DATA_BLOCK DB 5
AUTHOR : NUMERIK
FAMILY : _800D
NAME : Basics
VERSION : 1.5
  STRUCT
   Ch1_DB2_310 : BOOL  := TRUE;	// (Channel 1-10 ever 18 Bits):  error message
   Ch1_DB2_311 : BOOL ;	// Channel 1, DB2.DBB311; operational message
   Ch1_DB2_312 : BOOL  := TRUE;	// Channel 1, DB2.DBB312; error message
   Ch1_DB2_313 : BOOL  := TRUE;	// error message
   Ch1_DB2_314 : BOOL ;	// operational message
   Ch1_DB2_315 : BOOL ;	// operational message
   Ch1_DB2_316 : BOOL  := TRUE;	// error message
   Ch1_DB2_317 : BOOL  := TRUE;	// error message
   Ch1_DB2_318 : BOOL ;	// operational message
   Ch1_DB2_319 : BOOL ;	// operational message
   Ch1_DB2_320 : BOOL  := TRUE;	// error message
   Ch1_DB2_321 : BOOL ;	// operational message
   Ch1_DB2_322 : BOOL  := TRUE;	// error message
   Ch1_DB2_323 : BOOL ;	// operational message
   Ch1_DB2_324 : BOOL  := TRUE;	// error message
   Ch1_DB2_325 : BOOL ;	// operational message
   Ch1_DB2_326 : BOOL  := TRUE;	// error message
   Ch1_DB2_327 : BOOL ;	// operational message
   Ch2_DB2_328 : BOOL  := TRUE;	// Channel 2, DB2.DBB328; error message
   Ch2_DB2_329 : BOOL ;	// Channel 2, DB2.DBB329; operational message
   Ch2_DB2_330 : BOOL  := TRUE;	// error message
   Ch2_DB2_331 : BOOL  := TRUE;	// error message
   Ch2_DB2_332 : BOOL ;	// operational message
   Ch2_DB2_333 : BOOL ;	// operational message
   Ch2_DB2_334 : BOOL  := TRUE;	// error message
   Ch2_DB2_335 : BOOL  := TRUE;	// error message
   Ch2_DB2_336 : BOOL ;	// operational message
   Ch2_DB2_337 : BOOL ;	// operational message
   Ch2_DB2_338 : BOOL  := TRUE;	// error message
   Ch2_DB2_339 : BOOL ;	// operational message
   Ch2_DB2_340 : BOOL  := TRUE;	// error message
   Ch2_DB2_341 : BOOL ;	// operational message
   Ch2_DB2_342 : BOOL  := TRUE;	// error message
   Ch2_DB2_343 : BOOL ;	// operational message
   Ch2_DB2_344 : BOOL  := TRUE;	// error message
   Ch2_DB2_345 : BOOL ;	// operational message
   Ch3_DB2_346 : BOOL  := TRUE;	// Channel 3, DB2.DBB346; error message
   Ch3_DB2_347 : BOOL ;	// Channel 3, DB2.DBB347; operational message
   Ch3_DB2_348 : BOOL  := TRUE;	// error message
   Ch3_DB2_349 : BOOL  := TRUE;	// error message
   Ch3_DB2_350 : BOOL ;	// operational message
   Ch3_DB2_351 : BOOL ;	// operational message
   Ch3_DB2_352 : BOOL  := TRUE;	// error message
   Ch3_DB2_353 : BOOL  := TRUE;	// error message
   Ch3_DB2_354 : BOOL ;	// operational message
   Ch3_DB2_355 : BOOL ;	// operational message
   Ch3_DB2_356 : BOOL  := TRUE;	// error message
   Ch3_DB2_357 : BOOL ;	// operational message
   Ch3_DB2_358 : BOOL  := TRUE;	// error message
   Ch3_DB2_359 : BOOL ;	// operational message
   Ch3_DB2_360 : BOOL  := TRUE;	// error message
   Ch3_DB2_361 : BOOL ;	// operational message
   Ch3_DB2_362 : BOOL  := TRUE;	// error message
   Ch3_DB2_363 : BOOL ;	// operational message
   Ch4_DB2_364 : BOOL  := TRUE;	// Channel 4, DB2.DBB364; error message
   Ch4_DB2_365 : BOOL ;	// Channel 4, DB2.DBB365; operational message
   Ch4_DB2_366 : BOOL  := TRUE;	// error message
   Ch4_DB2_367 : BOOL  := TRUE;	// error message
   Ch4_DB2_368 : BOOL ;	// operational message
   Ch4_DB2_369 : BOOL ;	// operational message
   Ch4_DB2_370 : BOOL  := TRUE;	// error message
   Ch4_DB2_371 : BOOL  := TRUE;	// error message
   Ch4_DB2_372 : BOOL ;	// operational message
   Ch4_DB2_373 : BOOL ;	// operational message
   Ch4_DB2_374 : BOOL  := TRUE;	// error message
   Ch4_DB2_375 : BOOL ;	// operational message
   Ch4_DB2_376 : BOOL  := TRUE;	// error message
   Ch4_DB2_377 : BOOL ;	// operational message
   Ch4_DB2_378 : BOOL  := TRUE;	// error message
   Ch4_DB2_379 : BOOL ;	// operational message
   Ch4_DB2_380 : BOOL  := TRUE;	// error message
   Ch4_DB2_381 : BOOL ;	// operational message
   Ch5_DB2_382 : BOOL  := TRUE;	// Channel 5, DB2.DBB382; error message
   Ch5_DB2_383 : BOOL ;	// Channel 5, DB2.DBB383; operational message
   Ch5_DB2_384 : BOOL  := TRUE;	// error message
   Ch5_DB2_385 : BOOL  := TRUE;	// error message
   Ch5_DB2_386 : BOOL ;	// operational message
   Ch5_DB2_387 : BOOL ;	// operational message
   Ch5_DB2_388 : BOOL  := TRUE;	// error message
   Ch5_DB2_389 : BOOL  := TRUE;	// error message
   Ch5_DB2_390 : BOOL ;	// operational message
   Ch5_DB2_391 : BOOL ;	// operational message
   Ch5_DB2_392 : BOOL  := TRUE;	// error message
   Ch5_DB2_393 : BOOL ;	// operational message
   Ch5_DB2_394 : BOOL  := TRUE;	// error message
   Ch5_DB2_395 : BOOL ;	// operational message
   Ch5_DB2_396 : BOOL  := TRUE;	// error message
   Ch5_DB2_397 : BOOL ;	// operational message
   Ch5_DB2_398 : BOOL  := TRUE;	// error message
   Ch5_DB2_399 : BOOL ;	// operational message
   Ch6_DB2_400 : BOOL  := TRUE;	// Channel 6, DB2.DBB400; error message
   Ch6_DB2_401 : BOOL ;	// Channel 6, DB2.DBB401; operational message
   Ch6_DB2_402 : BOOL  := TRUE;	// error message
   Ch6_DB2_403 : BOOL  := TRUE;	// error message
   Ch6_DB2_404 : BOOL ;	// operational message
   Ch6_DB2_405 : BOOL ;	// operational message
   Ch6_DB2_406 : BOOL  := TRUE;	// error message
   Ch6_DB2_407 : BOOL  := TRUE;	// error message
   Ch6_DB2_408 : BOOL ;	// operational message
   Ch6_DB2_409 : BOOL ;	// operational message
   Ch6_DB2_410 : BOOL  := TRUE;	// error message
   Ch6_DB2_411 : BOOL ;	// operational message
   Ch6_DB2_412 : BOOL  := TRUE;	// error message
   Ch6_DB2_413 : BOOL ;	// operational message
   Ch6_DB2_414 : BOOL  := TRUE;	// error message
   Ch6_DB2_415 : BOOL ;	// operational message
   Ch6_DB2_416 : BOOL  := TRUE;	// error message
   Ch6_DB2_417 : BOOL ;	// operational message
   Ch7_DB2_418 : BOOL  := TRUE;	// Channel 7, DB2.DBB418; error message
   Ch7_DB2_419 : BOOL ;	// Channel 7, DB2.DBB419; operational message
   Ch7_DB2_420 : BOOL  := TRUE;	// error message
   Ch7_DB2_421 : BOOL  := TRUE;	// error message
   Ch7_DB2_422 : BOOL ;	// operational message
   Ch7_DB2_423 : BOOL ;	// operational message
   Ch7_DB2_424 : BOOL  := TRUE;	// error message
   Ch7_DB2_425 : BOOL  := TRUE;	// error message
   Ch7_DB2_426 : BOOL ;	// operational message
   Ch7_DB2_427 : BOOL ;	// operational message
   Ch7_DB2_428 : BOOL  := TRUE;	// error message
   Ch7_DB2_429 : BOOL ;	// operational message
   Ch7_DB2_430 : BOOL  := TRUE;	// error message
   Ch7_DB2_431 : BOOL ;	// operational message
   Ch7_DB2_432 : BOOL  := TRUE;	// error message
   Ch7_DB2_433 : BOOL ;	// operational message
   Ch7_DB2_434 : BOOL  := TRUE;	// error message
   Ch7_DB2_435 : BOOL ;	// operational message
   Ch8_DB2_436 : BOOL  := TRUE;	// Channel 8, DB2.DBB436; error message
   Ch8_DB2_437 : BOOL ;	// Channel 8, DB2.DBB437; operational message
   Ch8_DB2_438 : BOOL  := TRUE;	// error message
   Ch8_DB2_439 : BOOL  := TRUE;	// error message
   Ch8_DB2_440 : BOOL ;	// operational message
   Ch8_DB2_441 : BOOL ;	// operational message
   Ch8_DB2_442 : BOOL  := TRUE;	// error message
   Ch8_DB2_443 : BOOL  := TRUE;	// error message
   Ch8_DB2_444 : BOOL ;	// operational message
   Ch8_DB2_445 : BOOL ;	// operational message
   Ch8_DB2_446 : BOOL  := TRUE;	// error message
   Ch8_DB2_447 : BOOL ;	// operational message
   Ch8_DB2_448 : BOOL  := TRUE;	// error message
   Ch8_DB2_449 : BOOL ;	// operational message
   Ch8_DB2_450 : BOOL  := TRUE;	// error message
   Ch8_DB2_451 : BOOL ;	// operational message
   Ch8_DB2_452 : BOOL  := TRUE;	// error message
   Ch8_DB2_453 : BOOL ;	// operational message
   Ch9_DB2_454 : BOOL  := TRUE;	// Channel 9, DB2.DBB454; error message
   Ch9_DB2_455 : BOOL ;	// Channel 9, DB2.DBB455; operational message
   Ch9_DB2_456 : BOOL  := TRUE;	// error message
   Ch9_DB2_457 : BOOL  := TRUE;	// error message
   Ch9_DB2_458 : BOOL ;	// operational message
   Ch9_DB2_459 : BOOL ;	// operational message
   Ch9_DB2_460 : BOOL  := TRUE;	// error message
   Ch9_DB2_461 : BOOL  := TRUE;	// error message
   Ch9_DB2_462 : BOOL ;	// operational message
   Ch9_DB2_463 : BOOL ;	// operational message
   Ch9_DB2_464 : BOOL  := TRUE;	// error message
   Ch9_DB2_465 : BOOL ;	// operational message
   Ch9_DB2_466 : BOOL  := TRUE;	// error message
   Ch9_DB2_467 : BOOL ;	// operational message
   Ch9_DB2_468 : BOOL  := TRUE;	// error message
   Ch9_DB2_469 : BOOL ;	// operational message
   Ch9_DB2_470 : BOOL  := TRUE;	// error message
   Ch9_DB2_471 : BOOL ;	// operational message
   Ch10_DB2_472 : BOOL  := TRUE;	// Channel 10, DB2.DBB472; error message
   Ch10_DB2_473 : BOOL ;	// Channel 10, DB2.DBB473; operational message
   Ch10_DB2_474 : BOOL  := TRUE;	// error message
   Ch10_DB2_475 : BOOL  := TRUE;	// error message
   Ch10_DB2_476 : BOOL ;	// operational message
   Ch10_DB2_477 : BOOL ;	// operational message
   Ch10_DB2_478 : BOOL  := TRUE;	// error message
   Ch10_DB2_479 : BOOL  := TRUE;	// error message
   Ch10_DB2_480 : BOOL ;	// operational message
   Ch10_DB2_481 : BOOL ;	// operational message
   Ch10_DB2_482 : BOOL  := TRUE;	// error message
   Ch10_DB2_483 : BOOL ;	// operational message
   Ch10_DB2_484 : BOOL  := TRUE;	// error message
   Ch10_DB2_485 : BOOL ;	// operational message
   Ch10_DB2_486 : BOOL  := TRUE;	// error message
   Ch10_DB2_487 : BOOL ;	// operational message
   Ch10_DB2_488 : BOOL  := TRUE;	// error message
   Ch10_DB2_489 : BOOL ;	// operational message
   Ax1_DB2_490 : BOOL  := TRUE;	// (32 Axes/Spindles ever 2 Bit):  error message
   Ax1_DB2_491 : BOOL ;	// Axis 1, DB2.DBB491; operational message
   Ax2_DB2_492 : BOOL  := TRUE;	// Axis 2, DB2.DBB492; error message
   Ax2_DB2_493 : BOOL ;	// Axis 2, DB2.DBB493; operational message
   Ax3_DB2_494 : BOOL  := TRUE;	// error message
   Ax3_DB2_495 : BOOL ;	// operational message
   Ax4_DB2_496 : BOOL  := TRUE;	// error message
   Ax4_DB2_497 : BOOL ;	// operational message
   Ax5_DB2_498 : BOOL  := TRUE;	// error message
   Ax5_DB2_499 : BOOL ;	// operational message
   Ax6_DB2_500 : BOOL  := TRUE;	// error message
   Ax6_DB2_501 : BOOL ;	// operational message
   Ax7_DB2_502 : BOOL  := TRUE;	// error message
   Ax7_DB2_503 : BOOL ;	// operational message
   Ax8_DB2_504 : BOOL  := TRUE;	// error message
   Ax8_DB2_505 : BOOL ;	// operational message
   Ax9_DB2_506 : BOOL  := TRUE;	// error message
   Ax9_DB2_507 : BOOL ;	// operational message
   Ax10_DB2_508 : BOOL  := TRUE;	// error message
   Ax10_DB2_509 : BOOL ;	// operational message
   Ax11_DB2_510 : BOOL  := TRUE;	// error message
   Ax11_DB2_511 : BOOL ;	// operational message
   Ax12_DB2_512 : BOOL  := TRUE;	// error message
   Ax12_DB2_513 : BOOL ;	// operational message
   Ax13_DB2_514 : BOOL  := TRUE;	// error message
   Ax13_DB2_515 : BOOL ;	// operational message
   Ax14_DB2_516 : BOOL  := TRUE;	// error message
   Ax14_DB2_517 : BOOL ;	// operational message
   Ax15_DB2_518 : BOOL  := TRUE;	// error message
   Ax15_DB2_519 : BOOL ;	// operational message
   Ax16_DB2_520 : BOOL  := TRUE;	// error message
   Ax16_DB2_521 : BOOL ;	// operational message
   Ax17_DB2_522 : BOOL  := TRUE;	// error message
   Ax17_DB2_523 : BOOL ;	// operational message
   Ax18_DB2_524 : BOOL  := TRUE;	// error message
   Ax18_DB2_525 : BOOL ;	// operational message
   Ax19_DB2_526 : BOOL  := TRUE;	// error message
   Ax19_DB2_527 : BOOL ;	// operational message
   Ax20_DB2_528 : BOOL  := TRUE;	// error message
   Ax20_DB2_529 : BOOL ;	// operational message
   Ax21_DB2_530 : BOOL  := TRUE;	// error message
   Ax21_DB2_531 : BOOL ;	// operational message
   Ax22_DB2_532 : BOOL  := TRUE;	// error message
   Ax22_DB2_533 : BOOL ;	// operational message
   Ax23_DB2_534 : BOOL  := TRUE;	// error message
   Ax23_DB2_535 : BOOL ;	// operational message
   Ax24_DB2_536 : BOOL  := TRUE;	// error message
   Ax24_DB2_537 : BOOL ;	// operational message
   Ax25_DB2_538 : BOOL  := TRUE;	// error message
   Ax25_DB2_539 : BOOL ;	// operational message
   Ax26_DB2_540 : BOOL  := TRUE;	// error message
   Ax26_DB2_541 : BOOL ;	// operational message
   Ax27_DB2_542 : BOOL  := TRUE;	// error message
   Ax27_DB2_543 : BOOL ;	// operational message
   Ax28_DB2_544 : BOOL  := TRUE;	// error message
   Ax28_DB2_545 : BOOL ;	// operational message
   Ax29_DB2_546 : BOOL  := TRUE;	// error message
   Ax29_DB2_547 : BOOL ;	// operational message
   Ax30_DB2_548 : BOOL  := TRUE;	// error message
   Ax30_DB2_549 : BOOL ;	// operational message
   Ax31_DB2_550 : BOOL  := TRUE;	// error message
   Ax31_DB2_551 : BOOL ;	// operational message
   Ax32_DB2_552 : BOOL  := TRUE;	// error message
   Ax32_DB2_553 : BOOL ;	// operational message
   User0_DB2_554 : BOOL  := TRUE;	// (32 User data area ever 8 Bit):  error message
   User0_DB2_555 : BOOL  := TRUE;	// UserDataArea 0, DB2.DBB555; error message
   User0_DB2_556 : BOOL  := TRUE;	// error message
   User0_DB2_557 : BOOL  := TRUE;	// error message
   User0_DB2_558 : BOOL ;	// operational message
   User0_DB2_559 : BOOL ;	// operational message
   User0_DB2_560 : BOOL ;	// operational message
   User0_DB2_561 : BOOL ;	// operational message
   User1_DB2_562 : BOOL  := TRUE;	// UserDataArea 1, DB2.DBB562; error message
   User1_DB2_563 : BOOL  := TRUE;	// error message
   User1_DB2_564 : BOOL  := TRUE;	// error message
   User1_DB2_565 : BOOL  := TRUE;	// error message
   User1_DB2_566 : BOOL ;	// operational message
   User1_DB2_567 : BOOL ;	// operational message
   User1_DB2_568 : BOOL ;	// operational message
   User1_DB2_569 : BOOL ;	// operational message
   User2_DB2_570 : BOOL  := TRUE;	// UserDataArea 2, DB2.DBB570; error message
   User2_DB2_571 : BOOL  := TRUE;	// error message
   User2_DB2_572 : BOOL  := TRUE;	// error message
   User2_DB2_573 : BOOL  := TRUE;	// error message
   User2_DB2_574 : BOOL ;	// operational message
   User2_DB2_575 : BOOL ;	// operational message
   User2_DB2_576 : BOOL ;	// operational message
   User2_DB2_577 : BOOL ;	// operational message
   User3_DB2_578 : BOOL  := TRUE;	// UserDataArea 3, DB2.DBB578; error message
   User3_DB2_579 : BOOL  := TRUE;	// error message
   User3_DB2_580 : BOOL  := TRUE;	// error message
   User3_DB2_581 : BOOL  := TRUE;	// error message
   User3_DB2_582 : BOOL ;	// operational message
   User3_DB2_583 : BOOL ;	// operational message
   User3_DB2_584 : BOOL ;	// operational message
   User3_DB2_585 : BOOL ;	// operational message
   User4_DB2_586 : BOOL  := TRUE;	// UserDataArea 4, DB2.DBB586; error message
   User4_DB2_587 : BOOL  := TRUE;	// error message
   User4_DB2_588 : BOOL  := TRUE;	// error message
   User4_DB2_589 : BOOL  := TRUE;	// error message
   User4_DB2_590 : BOOL ;	// operational message
   User4_DB2_591 : BOOL ;	// operational message
   User4_DB2_592 : BOOL ;	// operational message
   User4_DB2_593 : BOOL ;	// operational message
   User5_DB2_594 : BOOL  := TRUE;	// UserDataArea 5, DB2.DBB594; error message
   User5_DB2_595 : BOOL  := TRUE;	// error message
   User5_DB2_596 : BOOL  := TRUE;	// error message
   User5_DB2_597 : BOOL  := TRUE;	// error message
   User5_DB2_598 : BOOL ;	// operational message
   User5_DB2_599 : BOOL ;	// operational message
   User5_DB2_600 : BOOL ;	// operational message
   User5_DB2_601 : BOOL ;	// operational message
   User6_DB2_602 : BOOL  := TRUE;	// UserDataArea 6, DB2.DBB602; error message
   User6_DB2_603 : BOOL  := TRUE;	// error message
   User6_DB2_604 : BOOL  := TRUE;	// error message
   User6_DB2_605 : BOOL  := TRUE;	// error message
   User6_DB2_606 : BOOL ;	// operational message
   User6_DB2_607 : BOOL ;	// operational message
   User6_DB2_608 : BOOL ;	// operational message
   User6_DB2_609 : BOOL ;	// operational message
   User7_DB2_610 : BOOL  := TRUE;	// UserDataArea 7, DB2.DBB610; error message
   User7_DB2_611 : BOOL  := TRUE;	// error message
   User7_DB2_612 : BOOL  := TRUE;	// error message
   User7_DB2_613 : BOOL  := TRUE;	// error message
   User7_DB2_614 : BOOL ;	// operational message
   User7_DB2_615 : BOOL ;	// operational message
   User7_DB2_616 : BOOL ;	// operational message
   User7_DB2_617 : BOOL ;	// operational message
   User8_DB2_618 : BOOL  := TRUE;	// UserDataArea 8, DB2.DBB618; error message
   User8_DB2_619 : BOOL  := TRUE;	// error message
   User8_DB2_620 : BOOL  := TRUE;	// error message
   User8_DB2_621 : BOOL  := TRUE;	// error message
   User8_DB2_622 : BOOL ;	// operational message
   User8_DB2_623 : BOOL ;	// operational message
   User8_DB2_624 : BOOL ;	// operational message
   User8_DB2_625 : BOOL ;	// operational message
   User9_DB2_626 : BOOL  := TRUE;	// UserDataArea 9, DB2.DBB626; error message
   User9_DB2_627 : BOOL  := TRUE;	// error message
   User9_DB2_628 : BOOL  := TRUE;	// error message
   User9_DB2_629 : BOOL  := TRUE;	// error message
   User9_DB2_630 : BOOL ;	// operational message
   User9_DB2_631 : BOOL ;	// operational message
   User9_DB2_632 : BOOL ;	// operational message
   User9_DB2_633 : BOOL ;	// operational message
   User10_DB2_634 : BOOL  := TRUE;	// UserDataArea 10, DB2.DBB634; error message
   User10_DB2_635 : BOOL  := TRUE;	// error message
   User10_DB2_636 : BOOL  := TRUE;	// error message
   User10_DB2_637 : BOOL  := TRUE;	// error message
   User10_DB2_638 : BOOL ;	// operational message
   User10_DB2_639 : BOOL ;	// operational message
   User10_DB2_640 : BOOL ;	// operational message
   User10_DB2_641 : BOOL ;	// operational message
   User11_DB2_642 : BOOL  := TRUE;	// UserDataArea 11, DB2.DBB642; error message
   User11_DB2_643 : BOOL  := TRUE;	// error message
   User11_DB2_644 : BOOL  := TRUE;	// error message
   User11_DB2_645 : BOOL  := TRUE;	// error message
   User11_DB2_646 : BOOL ;	// operational message
   User11_DB2_647 : BOOL ;	// operational message
   User11_DB2_648 : BOOL ;	// operational message
   User11_DB2_649 : BOOL ;	// operational message
   User12_DB2_650 : BOOL  := TRUE;	// UserDataArea 12, DB2.DBB650; error message
   User12_DB2_651 : BOOL  := TRUE;	// error message
   User12_DB2_652 : BOOL  := TRUE;	// error message
   User12_DB2_653 : BOOL  := TRUE;	// error message
   User12_DB2_654 : BOOL ;	// operational message
   User12_DB2_655 : BOOL ;	// operational message
   User12_DB2_656 : BOOL ;	// operational message
   User12_DB2_657 : BOOL ;	// operational message
   User13_DB2_658 : BOOL  := TRUE;	// UserDataArea 13, DB2.DBB658; error message
   User13_DB2_659 : BOOL  := TRUE;	// error message
   User13_DB2_660 : BOOL  := TRUE;	// error message
   User13_DB2_661 : BOOL  := TRUE;	// error message
   User13_DB2_662 : BOOL ;	// operational message
   User13_DB2_663 : BOOL ;	// operational message
   User13_DB2_664 : BOOL ;	// operational message
   User13_DB2_665 : BOOL ;	// operational message
   User14_DB2_666 : BOOL  := TRUE;	// UserDataArea 14, DB2.DBB666; error message
   User14_DB2_667 : BOOL  := TRUE;	// error message
   User14_DB2_668 : BOOL  := TRUE;	// error message
   User14_DB2_669 : BOOL  := TRUE;	// error message
   User14_DB2_670 : BOOL ;	// operational message
   User14_DB2_671 : BOOL ;	// operational message
   User14_DB2_672 : BOOL ;	// operational message
   User14_DB2_673 : BOOL ;	// operational message
   User15_DB2_674 : BOOL  := TRUE;	// UserDataArea 15, DB2.DBB674; error message
   User15_DB2_675 : BOOL  := TRUE;	// error message
   User15_DB2_676 : BOOL  := TRUE;	// error message
   User15_DB2_677 : BOOL  := TRUE;	// error message
   User15_DB2_678 : BOOL ;	// operational message
   User15_DB2_679 : BOOL ;	// operational message
   User15_DB2_680 : BOOL ;	// operational message
   User15_DB2_681 : BOOL ;	// operational message
   User16_DB2_682 : BOOL  := TRUE;	// UserDataArea 16, DB2.DBB682; error message
   User16_DB2_683 : BOOL  := TRUE;	// error message
   User16_DB2_684 : BOOL  := TRUE;	// error message
   User16_DB2_685 : BOOL  := TRUE;	// error message
   User16_DB2_686 : BOOL ;	// operational message
   User16_DB2_687 : BOOL ;	// operational message
   User16_DB2_688 : BOOL ;	// operational message
   User16_DB2_689 : BOOL ;	// operational message
   User17_DB2_690 : BOOL  := TRUE;	// UserDataArea 17, DB2.DBB690; error message
   User17_DB2_691 : BOOL  := TRUE;	// error message
   User17_DB2_692 : BOOL  := TRUE;	// error message
   User17_DB2_693 : BOOL  := TRUE;	// error message
   User17_DB2_694 : BOOL ;	// operational message
   User17_DB2_695 : BOOL ;	// operational message
   User17_DB2_696 : BOOL ;	// operational message
   User17_DB2_697 : BOOL ;	// operational message
   User18_DB2_698 : BOOL  := TRUE;	// UserDataArea 18, DB2.DBB698; error message
   User18_DB2_699 : BOOL  := TRUE;	// error message
   User18_DB2_700 : BOOL  := TRUE;	// error message
   User18_DB2_701 : BOOL  := TRUE;	// error message
   User18_DB2_702 : BOOL ;	// operational message
   User18_DB2_703 : BOOL ;	// operational message
   User18_DB2_704 : BOOL ;	// operational message
   User18_DB2_705 : BOOL ;	// operational message
   User19_DB2_706 : BOOL  := TRUE;	// UserDataArea 19, DB2.DBB706; error message
   User19_DB2_707 : BOOL  := TRUE;	// error message
   User19_DB2_708 : BOOL  := TRUE;	// error message
   User19_DB2_709 : BOOL  := TRUE;	// error message
   User19_DB2_710 : BOOL ;	// operational message
   User19_DB2_711 : BOOL ;	// operational message
   User19_DB2_712 : BOOL ;	// operational message
   User19_DB2_713 : BOOL ;	// operational message
   User20_DB2_714 : BOOL  := TRUE;	// UserDataArea 20, DB2.DBB714; error message
   User20_DB2_715 : BOOL  := TRUE;	// error message
   User20_DB2_716 : BOOL  := TRUE;	// error message
   User20_DB2_717 : BOOL  := TRUE;	// error message
   User20_DB2_718 : BOOL ;	// operational message
   User20_DB2_719 : BOOL ;	// operational message
   User20_DB2_720 : BOOL ;	// operational message
   User20_DB2_721 : BOOL ;	// operational message
   User21_DB2_722 : BOOL  := TRUE;	// UserDataArea 21, DB2.DBB722; error message
   User21_DB2_723 : BOOL  := TRUE;	// error message
   User21_DB2_724 : BOOL  := TRUE;	// error message
   User21_DB2_725 : BOOL  := TRUE;	// error message
   User21_DB2_726 : BOOL ;	// operational message
   User21_DB2_727 : BOOL ;	// operational message
   User21_DB2_728 : BOOL ;	// operational message
   User21_DB2_729 : BOOL ;	// operational message
   User22_DB2_730 : BOOL  := TRUE;	// UserDataArea 22, DB2.DBB730; error message
   User22_DB2_731 : BOOL  := TRUE;	// error message
   User22_DB2_732 : BOOL  := TRUE;	// error message
   User22_DB2_733 : BOOL  := TRUE;	// error message
   User22_DB2_734 : BOOL ;	// operational message
   User22_DB2_735 : BOOL ;	// operational message
   User22_DB2_736 : BOOL ;	// operational message
   User22_DB2_737 : BOOL ;	// operational message
   User23_DB2_738 : BOOL  := TRUE;	// UserDataArea 23, DB2.DBB738; error message
   User23_DB2_739 : BOOL  := TRUE;	// error message
   User23_DB2_740 : BOOL  := TRUE;	// error message
   User23_DB2_741 : BOOL  := TRUE;	// error message
   User23_DB2_742 : BOOL ;	// operational message
   User23_DB2_743 : BOOL ;	// operational message
   User23_DB2_744 : BOOL ;	// operational message
   User23_DB2_745 : BOOL ;	// operational message
   User24_DB2_746 : BOOL  := TRUE;	// UserDataArea 24, DB2.DBB746; error message
   User24_DB2_747 : BOOL  := TRUE;	// error message
   User24_DB2_748 : BOOL  := TRUE;	// error message
   User24_DB2_749 : BOOL  := TRUE;	// error message
   User24_DB2_750 : BOOL ;	// operational message
   User24_DB2_751 : BOOL ;	// operational message
   User24_DB2_752 : BOOL ;	// operational message
   User24_DB2_753 : BOOL ;	// operational message
   User25_DB2_754 : BOOL  := TRUE;	// UserDataArea 25, DB2.DBB754; error message
   User25_DB2_755 : BOOL  := TRUE;	// error message
   User25_DB2_756 : BOOL  := TRUE;	// error message
   User25_DB2_757 : BOOL  := TRUE;	// error message
   User25_DB2_758 : BOOL ;	// operational message
   User25_DB2_759 : BOOL ;	// operational message
   User25_DB2_760 : BOOL ;	// operational message
   User25_DB2_761 : BOOL ;	// operational message
   User26_DB2_762 : BOOL  := TRUE;	// UserDataArea 26, DB2.DBB762; error message
   User26_DB2_763 : BOOL  := TRUE;	// error message
   User26_DB2_764 : BOOL  := TRUE;	// error message
   User26_DB2_765 : BOOL  := TRUE;	// error message
   User26_DB2_766 : BOOL ;	// operational message
   User26_DB2_767 : BOOL ;	// operational message
   User26_DB2_768 : BOOL ;	// operational message
   User26_DB2_769 : BOOL ;	// operational message
   User27_DB2_770 : BOOL  := TRUE;	// UserDataArea 27, DB2.DBB770; error message
   User27_DB2_771 : BOOL  := TRUE;	// error message
   User27_DB2_772 : BOOL  := TRUE;	// error message
   User27_DB2_773 : BOOL  := TRUE;	// error message
   User27_DB2_774 : BOOL ;	// operational message
   User27_DB2_775 : BOOL ;	// operational message
   User27_DB2_776 : BOOL ;	// operational message
   User27_DB2_777 : BOOL ;	// operational message
   User28_DB2_778 : BOOL  := TRUE;	// UserDataArea 28, DB2.DBB778; error message
   User28_DB2_779 : BOOL  := TRUE;	// error message
   User28_DB2_780 : BOOL  := TRUE;	// error message
   User28_DB2_781 : BOOL  := TRUE;	// error message
   User28_DB2_782 : BOOL ;	// operational message
   User28_DB2_783 : BOOL ;	// operational message
   User28_DB2_784 : BOOL ;	// operational message
   User28_DB2_785 : BOOL ;	// operational message
   User29_DB2_786 : BOOL  := TRUE;	// UserDataArea 29, DB2.DBB786; error message
   User29_DB2_787 : BOOL  := TRUE;	// error message
   User29_DB2_788 : BOOL  := TRUE;	// error message
   User29_DB2_789 : BOOL  := TRUE;	// error message
   User29_DB2_790 : BOOL ;	// operational message
   User29_DB2_791 : BOOL ;	// operational message
   User29_DB2_792 : BOOL ;	// operational message
   User29_DB2_793 : BOOL ;	// operational message
   User30_DB2_794 : BOOL  := TRUE;	// UserDataArea 30, DB2.DBB794; error message
   User30_DB2_795 : BOOL  := TRUE;	// error message
   User30_DB2_796 : BOOL  := TRUE;	// error message
   User30_DB2_797 : BOOL  := TRUE;	// error message
   User30_DB2_798 : BOOL ;	// operational message
   User30_DB2_799 : BOOL ;	// operational message
   User30_DB2_800 : BOOL ;	// operational message
   User30_DB2_801 : BOOL ;	// operational message
   User31_DB2_802 : BOOL  := TRUE;	// UserDataArea 31, DB2.DBB802; error message
   User31_DB2_803 : BOOL  := TRUE;	// error message
   User31_DB2_804 : BOOL  := TRUE;	// error message
   User31_DB2_805 : BOOL  := TRUE;	// error message
   User31_DB2_806 : BOOL ;	// operational message
   User31_DB2_807 : BOOL ;	// operational message
   User31_DB2_808 : BOOL ;	// operational message
   User31_DB2_809 : BOOL ;	// operational message
   Bit62_4 : BOOL ;	// reserved
   Bit62_5 : BOOL ;	// reserved
   Bit62_6 : BOOL ;	// reserved
   Bit62_7 : BOOL ;	// reserved
   Byte63 : BYTE ;	// reserved
   Word64 : WORD ;	// reserved
   Word66 : WORD ;	// reserved
   Word68 : WORD ;	// reserved
   Word70 : WORD ;	// reserved
   UserDek2No : ARRAY  [0 .. 31 ] OF // UserDek2No: Value 0..9 possible
   BYTE  := B#16#0;
  END_STRUCT ;	
BEGIN
   Ch1_DB2_310 := TRUE;
   Ch1_DB2_312 := TRUE;
   Ch1_DB2_313 := TRUE;
   Ch1_DB2_316 := TRUE;
   Ch1_DB2_317 := TRUE;
   Ch1_DB2_320 := TRUE;
   Ch1_DB2_322 := TRUE;
   Ch1_DB2_324 := TRUE;
   Ch1_DB2_326 := TRUE;
   Ch2_DB2_328 := TRUE;
   Ch2_DB2_330 := TRUE;
   Ch2_DB2_331 := TRUE;
   Ch2_DB2_334 := TRUE;
   Ch2_DB2_335 := TRUE;
   Ch2_DB2_338 := TRUE;
   Ch2_DB2_340 := TRUE;
   Ch2_DB2_342 := TRUE;
   Ch2_DB2_344 := TRUE;
   Ch3_DB2_346 := TRUE;
   Ch3_DB2_348 := TRUE;
   Ch3_DB2_349 := TRUE;
   Ch3_DB2_352 := TRUE;
   Ch3_DB2_353 := TRUE;
   Ch3_DB2_356 := TRUE;
   Ch3_DB2_358 := TRUE;
   Ch3_DB2_360 := TRUE;
   Ch3_DB2_362 := TRUE;
   Ch4_DB2_364 := TRUE;
   Ch4_DB2_366 := TRUE;
   Ch4_DB2_367 := TRUE;
   Ch4_DB2_370 := TRUE;
   Ch4_DB2_371 := TRUE;
   Ch4_DB2_374 := TRUE;
   Ch4_DB2_376 := TRUE;
   Ch4_DB2_378 := TRUE;
   Ch4_DB2_380 := TRUE;
   Ch5_DB2_382 := TRUE;
   Ch5_DB2_384 := TRUE;
   Ch5_DB2_385 := TRUE;
   Ch5_DB2_388 := TRUE;
   Ch5_DB2_389 := TRUE;
   Ch5_DB2_392 := TRUE;
   Ch5_DB2_394 := TRUE;
   Ch5_DB2_396 := TRUE;
   Ch5_DB2_398 := TRUE;
   Ch6_DB2_400 := TRUE;
   Ch6_DB2_402 := TRUE;
   Ch6_DB2_403 := TRUE;
   Ch6_DB2_406 := TRUE;
   Ch6_DB2_407 := TRUE;
   Ch6_DB2_410 := TRUE;
   Ch6_DB2_412 := TRUE;
   Ch6_DB2_414 := TRUE;
   Ch6_DB2_416 := TRUE;
   Ch7_DB2_418 := TRUE;
   Ch7_DB2_420 := TRUE;
   Ch7_DB2_421 := TRUE;
   Ch7_DB2_424 := TRUE;
   Ch7_DB2_425 := TRUE;
   Ch7_DB2_428 := TRUE;
   Ch7_DB2_430 := TRUE;
   Ch7_DB2_432 := TRUE;
   Ch7_DB2_434 := TRUE;
   Ch8_DB2_436 := TRUE;
   Ch8_DB2_438 := TRUE;
   Ch8_DB2_439 := TRUE;
   Ch8_DB2_442 := TRUE;
   Ch8_DB2_443 := TRUE;
   Ch8_DB2_446 := TRUE;
   Ch8_DB2_448 := TRUE;
   Ch8_DB2_450 := TRUE;
   Ch8_DB2_452 := TRUE;
   Ch9_DB2_454 := TRUE;
   Ch9_DB2_456 := TRUE;
   Ch9_DB2_457 := TRUE;
   Ch9_DB2_460 := TRUE;
   Ch9_DB2_461 := TRUE;
   Ch9_DB2_464 := TRUE;
   Ch9_DB2_466 := TRUE;
   Ch9_DB2_468 := TRUE;
   Ch9_DB2_470 := TRUE;
   Ch10_DB2_472 := TRUE;
   Ch10_DB2_474 := TRUE;
   Ch10_DB2_475 := TRUE;
   Ch10_DB2_478 := TRUE;
   Ch10_DB2_479 := TRUE;
   Ch10_DB2_482 := TRUE;
   Ch10_DB2_484 := TRUE;
   Ch10_DB2_486 := TRUE;
   Ch10_DB2_488 := TRUE;
   Ax1_DB2_490 := TRUE;
   Ax2_DB2_492 := TRUE;
   Ax3_DB2_494 := TRUE;
   Ax4_DB2_496 := TRUE;
   Ax5_DB2_498 := TRUE;
   Ax6_DB2_500 := TRUE;
   Ax7_DB2_502 := TRUE;
   Ax8_DB2_504 := TRUE;
   Ax9_DB2_506 := TRUE;
   Ax10_DB2_508 := TRUE;
   Ax11_DB2_510 := TRUE;
   Ax12_DB2_512 := TRUE;
   Ax13_DB2_514 := TRUE;
   Ax14_DB2_516 := TRUE;
   Ax15_DB2_518 := TRUE;
   Ax16_DB2_520 := TRUE;
   Ax17_DB2_522 := TRUE;
   Ax18_DB2_524 := TRUE;
   Ax19_DB2_526 := TRUE;
   Ax20_DB2_528 := TRUE;
   Ax21_DB2_530 := TRUE;
   Ax22_DB2_532 := TRUE;
   Ax23_DB2_534 := TRUE;
   Ax24_DB2_536 := TRUE;
   Ax25_DB2_538 := TRUE;
   Ax26_DB2_540 := TRUE;
   Ax27_DB2_542 := TRUE;
   Ax28_DB2_544 := TRUE;
   Ax29_DB2_546 := TRUE;
   Ax30_DB2_548 := TRUE;
   Ax31_DB2_550 := TRUE;
   Ax32_DB2_552 := TRUE;
   User0_DB2_554 := TRUE;
   User0_DB2_555 := TRUE;
   User0_DB2_556 := TRUE;
   User0_DB2_557 := TRUE;
   User1_DB2_562 := TRUE;
   User1_DB2_563 := TRUE;
   User1_DB2_564 := TRUE;
   User1_DB2_565 := TRUE;
   User2_DB2_570 := TRUE;
   User2_DB2_571 := TRUE;
   User2_DB2_572 := TRUE;
   User2_DB2_573 := TRUE;
   User3_DB2_578 := TRUE;
   User3_DB2_579 := TRUE;
   User3_DB2_580 := TRUE;
   User3_DB2_581 := TRUE;
   User4_DB2_586 := TRUE;
   User4_DB2_587 := TRUE;
   User4_DB2_588 := TRUE;
   User4_DB2_589 := TRUE;
   User5_DB2_594 := TRUE;
   User5_DB2_595 := TRUE;
   User5_DB2_596 := TRUE;
   User5_DB2_597 := TRUE;
   User6_DB2_602 := TRUE;
   User6_DB2_603 := TRUE;
   User6_DB2_604 := TRUE;
   User6_DB2_605 := TRUE;
   User7_DB2_610 := TRUE;
   User7_DB2_611 := TRUE;
   User7_DB2_612 := TRUE;
   User7_DB2_613 := TRUE;
   User8_DB2_618 := TRUE;
   User8_DB2_619 := TRUE;
   User8_DB2_620 := TRUE;
   User8_DB2_621 := TRUE;
   User9_DB2_626 := TRUE;
   User9_DB2_627 := TRUE;
   User9_DB2_628 := TRUE;
   User9_DB2_629 := TRUE;
   User10_DB2_634 := TRUE;
   User10_DB2_635 := TRUE;
   User10_DB2_636 := TRUE;
   User10_DB2_637 := TRUE;
   User11_DB2_642 := TRUE;
   User11_DB2_643 := TRUE;
   User11_DB2_644 := TRUE;
   User11_DB2_645 := TRUE;
   User12_DB2_650 := TRUE;
   User12_DB2_651 := TRUE;
   User12_DB2_652 := TRUE;
   User12_DB2_653 := TRUE;
   User13_DB2_658 := TRUE;
   User13_DB2_659 := TRUE;
   User13_DB2_660 := TRUE;
   User13_DB2_661 := TRUE;
   User14_DB2_666 := TRUE;
   User14_DB2_667 := TRUE;
   User14_DB2_668 := TRUE;
   User14_DB2_669 := TRUE;
   User15_DB2_674 := TRUE;
   User15_DB2_675 := TRUE;
   User15_DB2_676 := TRUE;
   User15_DB2_677 := TRUE;
   User16_DB2_682 := TRUE;
   User16_DB2_683 := TRUE;
   User16_DB2_684 := TRUE;
   User16_DB2_685 := TRUE;
   User17_DB2_690 := TRUE;
   User17_DB2_691 := TRUE;
   User17_DB2_692 := TRUE;
   User17_DB2_693 := TRUE;
   User18_DB2_698 := TRUE;
   User18_DB2_699 := TRUE;
   User18_DB2_700 := TRUE;
   User18_DB2_701 := TRUE;
   User19_DB2_706 := TRUE;
   User19_DB2_707 := TRUE;
   User19_DB2_708 := TRUE;
   User19_DB2_709 := TRUE;
   User20_DB2_714 := TRUE;
   User20_DB2_715 := TRUE;
   User20_DB2_716 := TRUE;
   User20_DB2_717 := TRUE;
   User21_DB2_722 := TRUE;
   User21_DB2_723 := TRUE;
   User21_DB2_724 := TRUE;
   User21_DB2_725 := TRUE;
   User22_DB2_730 := TRUE;
   User22_DB2_731 := TRUE;
   User22_DB2_732 := TRUE;
   User22_DB2_733 := TRUE;
   User23_DB2_738 := TRUE;
   User23_DB2_739 := TRUE;
   User23_DB2_740 := TRUE;
   User23_DB2_741 := TRUE;
   User24_DB2_746 := TRUE;
   User24_DB2_747 := TRUE;
   User24_DB2_748 := TRUE;
   User24_DB2_749 := TRUE;
   User25_DB2_754 := TRUE;
   User25_DB2_755 := TRUE;
   User25_DB2_756 := TRUE;
   User25_DB2_757 := TRUE;
   User26_DB2_762 := TRUE;
   User26_DB2_763 := TRUE;
   User26_DB2_764 := TRUE;
   User26_DB2_765 := TRUE;
   User27_DB2_770 := TRUE;
   User27_DB2_771 := TRUE;
   User27_DB2_772 := TRUE;
   User27_DB2_773 := TRUE;
   User28_DB2_778 := TRUE;
   User28_DB2_779 := TRUE;
   User28_DB2_780 := TRUE;
   User28_DB2_781 := TRUE;
   User29_DB2_786 := TRUE;
   User29_DB2_787 := TRUE;
   User29_DB2_788 := TRUE;
   User29_DB2_789 := TRUE;
   User30_DB2_794 := TRUE;
   User30_DB2_795 := TRUE;
   User30_DB2_796 := TRUE;
   User30_DB2_797 := TRUE;
   User31_DB2_802 := TRUE;
   User31_DB2_803 := TRUE;
   User31_DB2_804 := TRUE;
   User31_DB2_805 := TRUE;
END_DATA_BLOCK

DATA_BLOCK "gp_par"	// DB 7
TITLE = Parameters for Baseprogram
AUTHOR : NUMERIK
FAMILY : _800D
NAME : Basics
VERSION : 1.5
"RUN_UP"
BEGIN
END_DATA_BLOCK

DATA_BLOCK DB 8
AUTHOR : NUMERIK
FAMILY : _800D
NAME : Basics
VERSION : 1.5
  STRUCT
   Fc19_1 : ARRAY  [0 .. 3 ] OF BYTE ;
   Res0 : ARRAY  [0 .. 3 ] OF BYTE ;
   plData : ARRAY  [8 .. 43 ] OF BYTE ;
   TestAuto : BYTE ;
   FirstCycle : BYTE ;
   Res4 : WORD ;
   Res5 : BYTE ;
   IsFb15Correct : BYTE ;
   Res6 : ARRAY  [50 .. 61 ] OF BYTE ;
   Fc19_2 : ARRAY  [0 .. 3 ] OF BYTE ;
   Res8 : ARRAY  [66 .. 81 ] OF BYTE ;
   S7_error_id : WORD ;
   S7_error_param : WORD ;
   S7_error_adr : DWORD ;
   MinCycleTime : INT ;
   AdaptTime : INT ;
   ActCycleTime : INT ;
  END_STRUCT ;	
BEGIN
END_DATA_BLOCK

DATA_BLOCK "NC"	// DB 10
VERSION : 0.1
  STRUCT
   A_Disabl_Inp1 : BOOL ;	//Disable digi. NCK input 1
   A_Disabl_Inp2 : BOOL ;	//Disable digi. NCK input 2
   A_Disabl_Inp3 : BOOL ;	//Disable digi. NCK input 3
   A_Disabl_Inp4 : BOOL ;	//Disable digi. NCK input 4
   A_Disabl_Inp5 : BOOL ;	//Disable digi. NCK input 5
   A_Disabl_Inp6 : BOOL ;	//Disable digi. NCK input 6
   A_Disabl_Inp7 : BOOL ;	//Disable digi. NCK input 7
   A_Disabl_Inp8 : BOOL ;	//Disable digi. NCK input 8
   A_Set_Inp1 : BOOL ;	//Set digi. NCK input 1
   A_Set_Inp2 : BOOL ;	//Set digi. NCK input 2
   A_Set_Inp3 : BOOL ;	//Set digi. NCK input 3
   A_Set_Inp4 : BOOL ;	//Set digi. NCK input 4
   A_Set_Inp5 : BOOL ;	//Set digi. NCK input 5
   A_Set_Inp6 : BOOL ;	//Set digi. NCK input 6
   A_Set_Inp7 : BOOL ;	//Set digi. NCK input 7
   A_Set_Inp8 : BOOL ;	//Set digi. NCK input 8
   f0_f15 : ARRAY  [0 .. 15 ] OF BOOL ;	//Reserved
   A_Disabl_Out1 : BOOL ;	//Disable digi. NCK output 1
   A_Disabl_Out2 : BOOL ;	//Disable digi. NCK output 2
   A_Disabl_Out3 : BOOL ;	//Disable digi. NCK output 3
   A_Disabl_Out4 : BOOL ;	//Disable digi. NCK output 4
   A_Disabl_Out5 : BOOL ;	//Disable digi. NCK output 5
   A_Disabl_Out6 : BOOL ;	//Disable digi. NCK output 6
   A_Disabl_Out7 : BOOL ;	//Disable digi. NCK output 7
   A_Disabl_Out8 : BOOL ;	//Disable digi. NCK output 8
   A_OvMask_Out1 : BOOL ;	//Overwrite mask of digi. output 1
   A_OvMask_Out2 : BOOL ;	//Overwrite mask of digi. output 2
   A_OvMask_Out3 : BOOL ;	//Overwrite mask of digi. output 3
   A_OvMask_Out4 : BOOL ;	//Overwrite mask of digi. output 4
   A_OvMask_Out5 : BOOL ;	//Overwrite mask of digi. output 5
   A_OvMask_Out6 : BOOL ;	//Overwrite mask of digi. output 6
   A_OvMask_Out7 : BOOL ;	//Overwrite mask of digi. output 7
   A_OvMask_Out8 : BOOL ;	//Overwrite mask of digi. output 8
   A_Set_Out1 : BOOL ;	//Set digi. NCK output 1
   A_Set_Out2 : BOOL ;	//Set digi. NCK output 2
   A_Set_Out3 : BOOL ;	//Set digi. NCK output 3
   A_Set_Out4 : BOOL ;	//Set digi. NCK output 4
   A_Set_Out5 : BOOL ;	//Set digi. NCK output 5
   A_Set_Out6 : BOOL ;	//Set digi. NCK output 6
   A_Set_Out7 : BOOL ;	//Set digi. NCK output 7
   A_Set_Out8 : BOOL ;	//Set digi. NCK output 8
   A_InMask_Out1 : BOOL ;	//Input mask of digi. output 1
   A_InMask_Out2 : BOOL ;	//Input mask of digi. output 2
   A_InMask_Out3 : BOOL ;	//Input mask of digi. output 3
   A_InMask_Out4 : BOOL ;	//Input mask of digi. output 4
   A_InMask_Out5 : BOOL ;	//Input mask of digi. output 5
   A_InMask_Out6 : BOOL ;	//Input mask of digi. output 6
   A_InMask_Out7 : BOOL ;	//Input mask of digi. output 7
   A_InMask_Out8 : BOOL ;	//Input mask of digi. output 8
   MCP1AxisTbl : ARRAY  [1 .. 22 ] OF BYTE  := B#16#1, B#16#2, B#16#3, B#16#4, B#16#5, B#16#6, B#16#7, B#16#8, B#16#9, B#16#A, B#16#B, B#16#C;	//Axis No. Table MCP1
   MCP1MaxAxis : WORD ;	//max. of Axisno, must be smaller or equal gp_par.MaxAxis
   MCP2AxisTbl : ARRAY  [1 .. 22 ] OF BYTE  := B#16#1, B#16#2, B#16#3, B#16#4, B#16#5, B#16#6, B#16#7, B#16#8, B#16#9, B#16#A, B#16#B, B#16#C;	//Axis No. Table MCP2
   MCP2MaxAxis : WORD ;	//max. of Axisno, must be smaller or equal gp_par.MaxAxis
   f56_0 : BOOL ;
   A_EMERGENCY : BOOL ;	//Emergency stop
   A_EMERGENCY_Ackn : BOOL ;	//Acknowledge emergency stop
   f56_3 : BOOL ;
   A_Keyswitch0 : BOOL ;	//Keyswitch position 0
   A_Keyswitch1 : BOOL ;	//Keyswitch position 1
   A_Keyswitch2 : BOOL ;	//Keyswitch position 2
   A_Keyswitch3 : BOOL ;	//Keyswitch position 3
   A_IncInModeGroup : BOOL ;	//INC inputs in mode group area active
   f57_1 : BOOL ;
   f57_2 : BOOL ;
   A_PCshutdown : BOOL ;	//PC shutdown 840Di
   f57_4 : BOOL ;
   f57_5 : BOOL ;
   f57_6 : BOOL ;
   f57_7 : BOOL ;
   A_CollCheckOff : BOOL ;	//Collisions Check Off
   f58_1 : BOOL ;
   f58_2 : BOOL ;
   f58_3 : BOOL ;
   f58_4 : BOOL ;
   f58_5 : BOOL ;
   f58_6 : BOOL ;
   f58_7 : BOOL ;
   f59 : BYTE ;
   E_ActVal_In1 : BOOL ;	//Actual value of digi. NCK input 1
   E_ActVal_In2 : BOOL ;	//Actual value of digi. NCK input 2
   E_ActVal_In3 : BOOL ;	//Actual value of digi. NCK input 3
   E_ActVal_In4 : BOOL ;	//Actual value of digi. NCK input 4
   f60_4 : BOOL ;
   f60_5 : BOOL ;
   f60_6 : BOOL ;
   f60_7 : BOOL ;
   f61_f62 : ARRAY  [61 .. 61 ] OF BYTE ;
   E_Setpoint_Out1 : BOOL ;	//Setpoint of digi. NCK output 1
   E_Setpoint_Out2 : BOOL ;	//Setpoint of digi. NCK output 2
   E_Setpoint_Out3 : BOOL ;	//Setpoint of digi. NCK output 3
   E_Setpoint_Out4 : BOOL ;	//Setpoint of digi. NCK output 4
   E_Setpoint_Out5 : BOOL ;	//Setpoint of digi. NCK output 5
   E_Setpoint_Out6 : BOOL ;	//Setpoint of digi. NCK output 6
   E_Setpoint_Out7 : BOOL ;	//Setpoint of digi. NCK output 7
   E_Setpoint_Out8 : BOOL ;	//Setpoint of digi. NCK output 8
   f65_f67 : ARRAY  [65 .. 66 ] OF BYTE ;
   E_HW1_moved : BYTE ;	//Handwheel 1 moved
   E_HW2_moved : BYTE ;	//Handwheel 2 moved
   E_HW3_moved : BYTE ;	//Handwheel 3 moved
   E_CounterInchMetr : BYTE ;	//Modification counter inch/metric system of units
   E_MCP1AxisValid : BOOL ;	//from HT6
   E_MCP1WCS : BOOL ;	//from HT6
   f72_2 : BOOL ;
   f72_3 : BOOL ;
   f72_4 : BOOL ;
   f72_5 : BOOL ;
   f72_6 : BOOL ;
   E_MCP1AxKeyDisp : BOOL ;	//Mcp1 Axis Key Displayed
   E_MCP2AxisValid : BOOL ;	//from HT6
   E_MCP2WCS : BOOL ;	//from HT6
   f73_2 : BOOL ;
   f73_3 : BOOL ;
   f73_4 : BOOL ;
   f73_5 : BOOL ;
   f73_6 : BOOL ;
   E_MCP2AxKeyDisp : BOOL ;	//Mcp2 Axis Key Displayed
   MCP1AxisFromHMI : ARRAY  [1 .. 6 ] OF BYTE ;	//Axistable from HT6
   MCP2AxisFromHMI : ARRAY  [1 .. 6 ] OF BYTE ;	//Axistable from HT6
   res86 : WORD ;
   res88 : BYTE ;
   res89 : BYTE ;
   epsToPlc : BYTE ;
   epsFromPlc : BYTE ;
   MpiDpOk : BOOL ;	//Slaves on MPI/DP Ok
   DpOk : BOOL ;	//Slaves on DP Ok
   f92_2 : BOOL ;
   f92_3 : BOOL ;
   f92_4 : BOOL ;
   f92_5 : BOOL ;
   f92_6 : BOOL ;
   f92_7 : BOOL ;
   f93 : BYTE ;
   f94 : BYTE ;
   f95 : BYTE ;
   f96_0 : BOOL ;
   f96_1 : BOOL ;
   f96_2 : BOOL ;
   f96_3 : BOOL ;
   f96_4 : BOOL ;
   f96_5 : BOOL ;
   f96_6 : BOOL ;
   f96_7 : BOOL ;
   E_Chan_HW1_A : BOOL ;	//Channel number for handwheel1 A
   E_Chan_HW1_B : BOOL ;	//Channel number for handwheel1 B
   E_Chan_HW1_C : BOOL ;	//Channel number for handwheel1 C
   E_Chan_HW1_D : BOOL ;	//Channel number for handwheel1 D
   f97_4 : BOOL ;
   f97_5 : BOOL ;
   f97_6 : BOOL ;
   f97_7 : BOOL ;
   E_Chan_HW2_A : BOOL ;	//Channel number for handwheel2 A
   E_Chan_HW2_B : BOOL ;	//Channel number for handwheel2 B
   E_Chan_HW2_C : BOOL ;	//Channel number for handwheel2 C
   E_Chan_HW2_D : BOOL ;	//Channel number for handwheel2 D
   f98_4 : BOOL ;
   f98_5 : BOOL ;
   f98_6 : BOOL ;
   f98_7 : BOOL ;
   E_Chan_HW3_A : BOOL ;	//Channel number for handwheel3 A
   E_Chan_HW3_B : BOOL ;	//Channel number for handwheel3 B
   E_Chan_HW3_C : BOOL ;	//Channel number for handwheel3 C
   E_Chan_HW3_D : BOOL ;	//Channel number for handwheel3 D
   f99_4 : BOOL ;
   f99_5 : BOOL ;
   f99_6 : BOOL ;
   f99_7 : BOOL ;
   E_Ax_A_HW1 : BOOL ;	//Axis number for handwheel1 A
   E_Ax_B_HW1 : BOOL ;	//Axis number for handwheel1 B
   E_Ax_C_HW1 : BOOL ;	//Axis number for handwheel1 C
   E_Ax_D_HW1 : BOOL ;	//Axis number for handwheel1 D
   E_Ax_E_HW1 : BOOL ;	//Axis number for handwheel1 E
   E_CHW_sel1 : BOOL ;	//Contour handwheel selected
   E_HW_sel1 : BOOL ;	//Handwheel selected
   E_Mach_Ax1 : BOOL ;	//Machine axis
   E_Ax_A_HW2 : BOOL ;	//Axis number for handwheel2 A
   E_Ax_B_HW2 : BOOL ;	//Axis number for handwheel2 B
   E_Ax_C_HW2 : BOOL ;	//Axis number for handwheel2 C
   E_Ax_D_HW2 : BOOL ;	//Axis number for handwheel2 D
   E_Ax_E_HW2 : BOOL ;	//Axis number for handwheel2 E
   E_CHW_sel2 : BOOL ;	//Contour handwheel selected
   E_HW_sel2 : BOOL ;	//Handwheel selected
   E_Mach_Ax2 : BOOL ;	//Machine axis
   E_Ax_A_HW3 : BOOL ;	//Axis number for handwheel3 A
   E_Ax_B_HW3 : BOOL ;	//Axis number for handwheel3 B
   E_Ax_C_HW3 : BOOL ;	//Axis number for handwheel3 C
   E_Ax_D_HW3 : BOOL ;	//Axis number for handwheel3 D
   E_Ax_E_HW3 : BOOL ;	//Axis number for handwheel3 E
   E_CHW_sel3 : BOOL ;	//Contour handwheel selected
   E_HW_sel3 : BOOL ;	//Handwheel selected
   E_Mach_Ax3 : BOOL ;	//Machine axis
   E_RemDiag : BOOL ;	//Remote Diagnostic
   f103_1 : BOOL ;
   f103_2 : BOOL ;
   f103_3 : BOOL ;
   f103_4 : BOOL ;
   E_ATready : BOOL ;	//AT-box ready
   E_MMCTemp : BOOL ;	//MMC temperature limit
   E_MMCBatt : BOOL ;	//MMC 101/102 battery alarm
   E_MCP1ready : BOOL ;	//MCP1 ready;
   E_MCP2ready : BOOL ;	//MCP2 ready;
   E_BHGready : BOOL ;	//BHG ready;
   f104_3 : BOOL ;
   f104_4 : BOOL ;
   f104_5 : BOOL ;
   E_FirstOB1 : BOOL ;	//This bit is on for the first OB1 cycle
   E_NCKready : BOOL ;	//NCK CPU ready
   f105 : BYTE ;
   E_CollCheckOff : BOOL ;	//CollisionsCheck Off
   E_EMSTOP : BOOL ;	//EMERGENCY STOP active
   f106_2 : BOOL ;
   f106_3 : BOOL ;
   f106_4 : BOOL ;
   f106_5 : BOOL ;
   f106_6 : BOOL ;
   f106_7 : BOOL ;
   E_InspProbe1 : BOOL ;	//Inspection probe 1 actuated
   E_InspProbe2 : BOOL ;	//Inspection probe 2 actuated
   f107_2 : BOOL ;
   f107_3 : BOOL ;
   f107_4 : BOOL ;
   f107_5 : BOOL ;
   E_NCU_LinkActive : BOOL ;	//NCU link active
   E_SystemInchDim : BOOL ;	//System inch dimension
   f108_0 : BOOL ;
   E_MMC2Ready : BOOL ;	//MMC2-CPU ready
   E_MMCMPIready : BOOL ;	//MMC1-CPU on MPI ready
   E_MMCBTSSready : BOOL ;	//MMC1-CPU on BTSS ready
   f108_4 : BOOL ;
   E_DrivesInCylOp : BOOL ;	//Drives in cylindric operation
   E_611Dready : BOOL ;	//611D ready
   E_NCready : BOOL ;
   E_NCKalarm : BOOL ;	//NCK alarm present
   f109_1 : BOOL ;
   f109_2 : BOOL ;
   f109_3 : BOOL ;
   A_PC_OSfault : BOOL ;	//PC operating system fault, 840Di
   E_HTempAlarm : BOOL ;	//Heat sink temperature alarm NCU 573
   E_ATempAlarm : BOOL ;	//Air temperature alarm
   E_BattAlarm : BOOL ;	//NCK battery alarm
   E_SWCamMinus : ARRAY  [0 .. 31 ] OF BOOL ;	//Software cams minus [0..31]
   E_SWCamPlus : ARRAY  [0 .. 31 ] OF BOOL ;	//Software cams plus [0..31]
   f118_f121 : ARRAY  [0 .. 3 ] OF BYTE ;
   A_Disabl_Inp9 : BOOL ;	//Disable digi. NCK input 9
   A_Disabl_Inp10 : BOOL ;	//Disable digi. NCK input 10
   A_Disabl_Inp11 : BOOL ;	//Disable digi. NCK input 11
   A_Disabl_Inp12 : BOOL ;	//Disable digi. NCK input 12
   A_Disabl_Inp13 : BOOL ;	//Disable digi. NCK input 13
   A_Disabl_Inp14 : BOOL ;	//Disable digi. NCK input 14
   A_Disabl_Inp15 : BOOL ;	//Disable digi. NCK input 15
   A_Disabl_Inp16 : BOOL ;	//Disable digi. NCK input 16
   A_Set_Inp9 : BOOL ;	//Set digi. NCK input 9
   A_Set_Inp10 : BOOL ;	//Set digi. NCK input 10
   A_Set_Inp11 : BOOL ;	//Set digi. NCK input 11
   A_Set_Inp12 : BOOL ;	//Set digi. NCK input 12
   A_Set_Inp13 : BOOL ;	//Set digi. NCK input 13
   A_Set_Inp14 : BOOL ;	//Set digi. NCK input 14
   A_Set_Inp15 : BOOL ;	//Set digi. NCK input 15
   A_Set_Inp16 : BOOL ;	//Set digi. NCK input 16
   A_Disabl_Inp17 : BOOL ;	//Disable digi. NCK input 17
   A_Disabl_Inp18 : BOOL ;	//Disable digi. NCK input 18
   A_Disabl_Inp19 : BOOL ;	//Disable digi. NCK input 19
   A_Disabl_Inp20 : BOOL ;	//Disable digi. NCK input 20
   A_Disabl_Inp21 : BOOL ;	//Disable digi. NCK input 21
   A_Disabl_Inp22 : BOOL ;	//Disable digi. NCK input 22
   A_Disabl_Inp23 : BOOL ;	//Disable digi. NCK input 23
   A_Disabl_Inp24 : BOOL ;	//Disable digi. NCK input 24
   A_Set_Inp17 : BOOL ;	//Set digi. NCK input 17
   A_Set_Inp18 : BOOL ;	//Set digi. NCK input 18
   A_Set_Inp19 : BOOL ;	//Set digi. NCK input 19
   A_Set_Inp20 : BOOL ;	//Set digi. NCK input 20
   A_Set_Inp21 : BOOL ;	//Set digi. NCK input 21
   A_Set_Inp22 : BOOL ;	//Set digi. NCK input 22
   A_Set_Inp23 : BOOL ;	//Set digi. NCK input 23
   A_Set_Inp24 : BOOL ;	//Set digi. NCK input 24
   A_Disabl_Inp25 : BOOL ;	//Disable digi. NCK input 25
   A_Disabl_Inp26 : BOOL ;	//Disable digi. NCK input 26
   A_Disabl_Inp27 : BOOL ;	//Disable digi. NCK input 27
   A_Disabl_Inp28 : BOOL ;	//Disable digi. NCK input 28
   A_Disabl_Inp29 : BOOL ;	//Disable digi. NCK input 29
   A_Disabl_Inp30 : BOOL ;	//Disable digi. NCK input 30
   A_Disabl_Inp31 : BOOL ;	//Disable digi. NCK input 31
   A_Disabl_Inp32 : BOOL ;	//Disable digi. NCK input 32
   A_Set_Inp25 : BOOL ;	//Set digi. NCK input 25
   A_Set_Inp26 : BOOL ;	//Set digi. NCK input 26
   A_Set_Inp27 : BOOL ;	//Set digi. NCK input 27
   A_Set_Inp28 : BOOL ;	//Set digi. NCK input 28
   A_Set_Inp29 : BOOL ;	//Set digi. NCK input 29
   A_Set_Inp30 : BOOL ;	//Set digi. NCK input 30
   A_Set_Inp31 : BOOL ;	//Set digi. NCK input 31
   A_Set_Inp32 : BOOL ;	//Set digi. NCK input 32
   A_Disabl_Inp33 : BOOL ;	//Disable digi. NCK input 33
   A_Disabl_Inp34 : BOOL ;	//Disable digi. NCK input 34
   A_Disabl_Inp35 : BOOL ;	//Disable digi. NCK input 35
   A_Disabl_Inp36 : BOOL ;	//Disable digi. NCK input 36
   A_Disabl_Inp37 : BOOL ;	//Disable digi. NCK input 37
   A_Disabl_Inp38 : BOOL ;	//Disable digi. NCK input 38
   A_Disabl_Inp39 : BOOL ;	//Disable digi. NCK input 39
   A_Disabl_Inp40 : BOOL ;	//Disable digi. NCK input 40
   A_Set_Inp33 : BOOL ;	//Set digi. NCK input 33
   A_Set_Inp34 : BOOL ;	//Set digi. NCK input 34
   A_Set_Inp35 : BOOL ;	//Set digi. NCK input 35
   A_Set_Inp36 : BOOL ;	//Set digi. NCK input 36
   A_Set_Inp37 : BOOL ;	//Set digi. NCK input 37
   A_Set_Inp38 : BOOL ;	//Set digi. NCK input 38
   A_Set_Inp39 : BOOL ;	//Set digi. NCK input 39
   A_Set_Inp40 : BOOL ;	//Set digi. NCK input 40
   A_Disabl_Out9 : BOOL ;	//Disable digi. NCK output 9
   A_Disabl_Out10 : BOOL ;	//Disable digi. NCK output 10
   A_Disabl_Out11 : BOOL ;	//Disable digi. NCK output 11
   A_Disabl_Out12 : BOOL ;	//Disable digi. NCK output 12
   A_Disabl_Out13 : BOOL ;	//Disable digi. NCK output 13
   A_Disabl_Out14 : BOOL ;	//Disable digi. NCK output 14
   A_Disabl_Out15 : BOOL ;	//Disable digi. NCK output 15
   A_Disabl_Out16 : BOOL ;	//Disable digi. NCK output 16
   A_OvMask_Out9 : BOOL ;	//Overwrite mask of digi. output 9
   A_OvMask_Out10 : BOOL ;	//Overwrite mask of digi. output 10
   A_OvMask_Out11 : BOOL ;	//Overwrite mask of digi. output 11
   A_OvMask_Out12 : BOOL ;	//Overwrite mask of digi. output 12
   A_OvMask_Out13 : BOOL ;	//Overwrite mask of digi. output 13
   A_OvMask_Out14 : BOOL ;	//Overwrite mask of digi. output 14
   A_OvMask_Out15 : BOOL ;	//Overwrite mask of digi. output 15
   A_OvMask_Out16 : BOOL ;	//Overwrite mask of digi. output 16
   A_Setval_Out9 : BOOL ;	//Set value digi. NCK output 9
   A_Setval_Out10 : BOOL ;	//Set value digi. NCK output 10
   A_Setval_Out11 : BOOL ;	//Set value digi. NCK output 11
   A_Setval_Out12 : BOOL ;	//Set value digi. NCK output 12
   A_Setval_Out13 : BOOL ;	//Set value digi. NCK output 13
   A_Setval_Out14 : BOOL ;	//Set value digi. NCK output 14
   A_Setval_Out15 : BOOL ;	//Set value digi. NCK output 15
   A_Setval_Out16 : BOOL ;	//Set value digi. NCK output 16
   A_InMask_Out9 : BOOL ;	//Input mask of digi. output 9
   A_InMask_Out10 : BOOL ;	//Input mask of digi. output 10
   A_InMask_Out11 : BOOL ;	//Input mask of digi. output 11
   A_InMask_Out12 : BOOL ;	//Input mask of digi. output 12
   A_InMask_Out13 : BOOL ;	//Input mask of digi. output 13
   A_InMask_Out14 : BOOL ;	//Input mask of digi. output 14
   A_InMask_Out15 : BOOL ;	//Input mask of digi. output 15
   A_InMask_Out16 : BOOL ;	//Input mask of digi. output 16
   A_Disabl_Out17 : BOOL ;	//Disable digi. NCK output 17
   A_Disabl_Out18 : BOOL ;	//Disable digi. NCK output 18
   A_Disabl_Out19 : BOOL ;	//Disable digi. NCK output 19
   A_Disabl_Out20 : BOOL ;	//Disable digi. NCK output 20
   A_Disabl_Out21 : BOOL ;	//Disable digi. NCK output 21
   A_Disabl_Out22 : BOOL ;	//Disable digi. NCK output 22
   A_Disabl_Out23 : BOOL ;	//Disable digi. NCK output 23
   A_Disabl_Out24 : BOOL ;	//Disable digi. NCK output 24
   A_OvMask_Out17 : BOOL ;	//Overwrite mask of digi. output 17
   A_OvMask_Out18 : BOOL ;	//Overwrite mask of digi. output 18
   A_OvMask_Out19 : BOOL ;	//Overwrite mask of digi. output 19
   A_OvMask_Out20 : BOOL ;	//Overwrite mask of digi. output 20
   A_OvMask_Out21 : BOOL ;	//Overwrite mask of digi. output 21
   A_OvMask_Out22 : BOOL ;	//Overwrite mask of digi. output 22
   A_OvMask_Out23 : BOOL ;	//Overwrite mask of digi. output 23
   A_OvMask_Out24 : BOOL ;	//Overwrite mask of digi. output 24
   A_Setval_Out17 : BOOL ;	//Set value digi. NCK output 17
   A_Setval_Out18 : BOOL ;	//Set value digi. NCK output 18
   A_Setval_Out19 : BOOL ;	//Set value digi. NCK output 19
   A_Setval_Out20 : BOOL ;	//Set value digi. NCK output 20
   A_Setval_Out21 : BOOL ;	//Set value digi. NCK output 21
   A_Setval_Out22 : BOOL ;	//Set value digi. NCK output 22
   A_Setval_Out23 : BOOL ;	//Set value digi. NCK output 23
   A_Setval_Out24 : BOOL ;	//Set value digi. NCK output 24
   A_InMask_Out17 : BOOL ;	//Input mask of digi. output 17
   A_InMask_Out18 : BOOL ;	//Input mask of digi. output 18
   A_InMask_Out19 : BOOL ;	//Input mask of digi. output 19
   A_InMask_Out20 : BOOL ;	//Input mask of digi. output 20
   A_InMask_Out21 : BOOL ;	//Input mask of digi. output 21
   A_InMask_Out22 : BOOL ;	//Input mask of digi. output 22
   A_InMask_Out23 : BOOL ;	//Input mask of digi. output 23
   A_InMask_Out24 : BOOL ;	//Input mask of digi. output 24
   A_Disabl_Out25 : BOOL ;	//Disable digi. NCK output 25
   A_Disabl_Out26 : BOOL ;	//Disable digi. NCK output 26
   A_Disabl_Out27 : BOOL ;	//Disable digi. NCK output 27
   A_Disabl_Out28 : BOOL ;	//Disable digi. NCK output 28
   A_Disabl_Out29 : BOOL ;	//Disable digi. NCK output 29
   A_Disabl_Out30 : BOOL ;	//Disable digi. NCK output 30
   A_Disabl_Out31 : BOOL ;	//Disable digi. NCK output 31
   A_Disabl_Out32 : BOOL ;	//Disable digi. NCK output 32
   A_OvMask_Out25 : BOOL ;	//Overwrite mask of digi. output 25
   A_OvMask_Out26 : BOOL ;	//Overwrite mask of digi. output 26
   A_OvMask_Out27 : BOOL ;	//Overwrite mask of digi. output 27
   A_OvMask_Out28 : BOOL ;	//Overwrite mask of digi. output 28
   A_OvMask_Out29 : BOOL ;	//Overwrite mask of digi. output 29
   A_OvMask_Out30 : BOOL ;	//Overwrite mask of digi. output 30
   A_OvMask_Out31 : BOOL ;	//Overwrite mask of digi. output 31
   A_OvMask_Out32 : BOOL ;	//Overwrite mask of digi. output 32
   A_Setval_Out25 : BOOL ;	//Set value digi. NCK output 25
   A_Setval_Out26 : BOOL ;	//Set value digi. NCK output 26
   A_Setval_Out27 : BOOL ;	//Set value digi. NCK output 27
   A_Setval_Out28 : BOOL ;	//Set value digi. NCK output 28
   A_Setval_Out29 : BOOL ;	//Set value digi. NCK output 29
   A_Setval_Out30 : BOOL ;	//Set value digi. NCK output 30
   A_Setval_Out31 : BOOL ;	//Set value digi. NCK output 31
   A_Setval_Out32 : BOOL ;	//Set value digi. NCK output 32
   A_InMask_Out25 : BOOL ;	//Input mask of digi. output 25
   A_InMask_Out26 : BOOL ;	//Input mask of digi. output 26
   A_InMask_Out27 : BOOL ;	//Input mask of digi. output 27
   A_InMask_Out28 : BOOL ;	//Input mask of digi. output 28
   A_InMask_Out29 : BOOL ;	//Input mask of digi. output 29
   A_InMask_Out30 : BOOL ;	//Input mask of digi. output 30
   A_InMask_Out31 : BOOL ;	//Input mask of digi. output 31
   A_InMask_Out32 : BOOL ;	//Input mask of digi. output 32
   A_Disabl_Out33 : BOOL ;	//Disable digi. NCK output 33
   A_Disabl_Out34 : BOOL ;	//Disable digi. NCK output 34
   A_Disabl_Out35 : BOOL ;	//Disable digi. NCK output 35
   A_Disabl_Out36 : BOOL ;	//Disable digi. NCK output 36
   A_Disabl_Out37 : BOOL ;	//Disable digi. NCK output 37
   A_Disabl_Out38 : BOOL ;	//Disable digi. NCK output 38
   A_Disabl_Out39 : BOOL ;	//Disable digi. NCK output 39
   A_Disabl_Out40 : BOOL ;	//Disable digi. NCK output 40
   A_OvMask_Out33 : BOOL ;	//Overwrite mask of digi. output 33
   A_OvMask_Out34 : BOOL ;	//Overwrite mask of digi. output 34
   A_OvMask_Out35 : BOOL ;	//Overwrite mask of digi. output 35
   A_OvMask_Out36 : BOOL ;	//Overwrite mask of digi. output 36
   A_OvMask_Out37 : BOOL ;	//Overwrite mask of digi. output 37
   A_OvMask_Out38 : BOOL ;	//Overwrite mask of digi. output 38
   A_OvMask_Out39 : BOOL ;	//Overwrite mask of digi. output 39
   A_OvMask_Out40 : BOOL ;	//Overwrite mask of digi. output 40
   A_Setval_out33 : BOOL ;	//Set value digi. NCK output 33
   A_Setval_out34 : BOOL ;	//Set value digi. NCK output 34
   A_Setval_out35 : BOOL ;	//Set value digi. NCK output 35
   A_Setval_out36 : BOOL ;	//Set value digi. NCK output 36
   A_Setval_out37 : BOOL ;	//Set value digi. NCK output 37
   A_Setval_out38 : BOOL ;	//Set value digi. NCK output 38
   A_Setval_out39 : BOOL ;	//Set value digi. NCK output 39
   A_Setval_out40 : BOOL ;	//Set value digi. NCK output 40
   A_InMask_Out33 : BOOL ;	//Input mask of digi. output 33
   A_InMask_Out34 : BOOL ;	//Input mask of digi. output 34
   A_InMask_Out35 : BOOL ;	//Input mask of digi. output 35
   A_InMask_Out36 : BOOL ;	//Input mask of digi. output 36
   A_InMask_Out37 : BOOL ;	//Input mask of digi. output 37
   A_InMask_Out38 : BOOL ;	//Input mask of digi. output 38
   A_InMask_Out39 : BOOL ;	//Input mask of digi. output 39
   A_InMask_Out40 : BOOL ;	//Input mask of digi. output 40
   A_Disabl_anaIn1 : BOOL ;	//Disable analog NCK input 1
   A_Disabl_anaIn2 : BOOL ;	//Disable analog NCK input 2
   A_Disabl_anaIn3 : BOOL ;	//Disable analog NCK input 3
   A_Disabl_anaIn4 : BOOL ;	//Disable analog NCK input 4
   A_Disabl_anaIn5 : BOOL ;	//Disable analog NCK input 5
   A_Disabl_anaIn6 : BOOL ;	//Disable analog NCK input 6
   A_Disabl_anaIn7 : BOOL ;	//Disable analog NCK input 7
   A_Disabl_anaIn8 : BOOL ;	//Disable analog NCK input 8
   A_InMask_anaIn1 : BOOL ;	//Input mask of analog NCK input 1
   A_InMask_anaIn2 : BOOL ;	//Input mask of analog NCK input 2
   A_InMask_anaIn3 : BOOL ;	//Input mask of analog NCK input 3
   A_InMask_anaIn4 : BOOL ;	//Input mask of analog NCK input 4
   A_InMask_anaIn5 : BOOL ;	//Input mask of analog NCK input 5
   A_InMask_anaIn6 : BOOL ;	//Input mask of analog NCK input 6
   A_InMask_anaIn7 : BOOL ;	//Input mask of analog NCK input 7
   A_InMask_anaIn8 : BOOL ;	//Input mask of analog NCK input 8
   A_Setval_anaIn1 : WORD ;	//Set value of analog NCK input 1
   A_Setval_anaIn2 : WORD ;	//Set value of analog NCK input 2
   A_Setval_anaIn3 : WORD ;	//Set value of analog NCK input 3
   A_Setval_anaIn4 : WORD ;	//Set value of analog NCK input 4
   A_Setval_anaIn5 : WORD ;	//Set value of analog NCK input 5
   A_Setval_anaIn6 : WORD ;	//Set value of analog NCK input 6
   A_Setval_anaIn7 : WORD ;	//Set value of analog NCK input 7
   A_Setval_anaIn8 : WORD ;	//Set value of analog NCK input 8
   f164_f165 : INT ;
   A_OvMask_anaOut1 : BOOL ;	//Overwrite mask of analog output 1
   A_OvMask_anaOut2 : BOOL ;	//Overwrite mask of analog output 2
   A_OvMask_anaOut3 : BOOL ;	//Overwrite mask of analog output 3
   A_OvMask_anaOut4 : BOOL ;	//Overwrite mask of analog output 4
   A_OvMask_anaOut5 : BOOL ;	//Overwrite mask of analog output 5
   A_OvMask_anaOut6 : BOOL ;	//Overwrite mask of analog output 6
   A_OvMask_anaOut7 : BOOL ;	//Overwrite mask of analog output 7
   A_OvMask_anaOut8 : BOOL ;	//Overwrite mask of analog output 8
   A_InMask_anaOut1 : BOOL ;	//Input mask of analog NCK output 1
   A_InMask_anaOut2 : BOOL ;	//Input mask of analog NCK output 2
   A_InMask_anaOut3 : BOOL ;	//Input mask of analog NCK output 3
   A_InMask_anaOut4 : BOOL ;	//Input mask of analog NCK output 4
   A_InMask_anaOut5 : BOOL ;	//Input mask of analog NCK output 5
   A_InMask_anaOut6 : BOOL ;	//Input mask of analog NCK output 6
   A_InMask_anaOut7 : BOOL ;	//Input mask of analog NCK output 7
   A_InMask_anaOut8 : BOOL ;	//Input mask of analog NCK output 8
   A_Disabl_anaOut1 : BOOL ;	//Disable analog NCK output 1
   A_Disabl_anaOut2 : BOOL ;	//Disable analog NCK output 2
   A_Disabl_anaOut3 : BOOL ;	//Disable analog NCK output 3
   A_Disabl_anaOut4 : BOOL ;	//Disable analog NCK output 4
   A_Disabl_anaOut5 : BOOL ;	//Disable analog NCK output 5
   A_Disabl_anaOut6 : BOOL ;	//Disable analog NCK output 6
   A_Disabl_anaOut7 : BOOL ;	//Disable analog NCK output 7
   A_Disabl_anaOut8 : BOOL ;	//Disable analog NCK output 8
   f169 : BYTE ;
   A_Setval_anaOut1 : WORD ;	//Set value of analog NCK output 1
   A_Setval_anaOut2 : WORD ;	//Set value of analog NCK output 2
   A_Setval_anaOut3 : WORD ;	//Set value of analog NCK output 3
   A_Setval_anaOut4 : WORD ;	//Set value of analog NCK output 4
   A_Setval_anaOut5 : WORD ;	//Set value of analog NCK output 5
   A_Setval_anaOut6 : WORD ;	//Set value of analog NCK output 6
   A_Setval_anaOut7 : WORD ;	//Set value of analog NCK output 7
   A_Setval_anaOut8 : WORD ;	//Set value of analog NCK output 8
   E_ActVal_In9 : BOOL ;	//Actual value of digi. NCK input 9
   E_ActVal_In10 : BOOL ;	//Actual value of digi. NCK input 10
   E_ActVal_In11 : BOOL ;	//Actual value of digi. NCK input 11
   E_ActVal_In12 : BOOL ;	//Actual value of digi. NCK input 12
   E_ActVal_In13 : BOOL ;	//Actual value of digi. NCK input 13
   E_ActVal_In14 : BOOL ;	//Actual value of digi. NCK input 14
   E_ActVal_In15 : BOOL ;	//Actual value of digi. NCK input 15
   E_ActVal_In16 : BOOL ;	//Actual value of digi. NCK input 16
   E_ActVal_In17 : BOOL ;	//Actual value of digi. NCK input 17
   E_ActVal_In18 : BOOL ;	//Actual value of digi. NCK input 18
   E_ActVal_In19 : BOOL ;	//Actual value of digi. NCK input 19
   E_ActVal_In20 : BOOL ;	//Actual value of digi. NCK input 20
   E_ActVal_In21 : BOOL ;	//Actual value of digi. NCK input 21
   E_ActVal_In22 : BOOL ;	//Actual value of digi. NCK input 22
   E_ActVal_In23 : BOOL ;	//Actual value of digi. NCK input 23
   E_ActVal_In24 : BOOL ;	//Actual value of digi. NCK input 24
   E_ActVal_In25 : BOOL ;	//Actual value of digi. NCK input 25
   E_ActVal_In26 : BOOL ;	//Actual value of digi. NCK input 26
   E_ActVal_In27 : BOOL ;	//Actual value of digi. NCK input 27
   E_ActVal_In28 : BOOL ;	//Actual value of digi. NCK input 28
   E_ActVal_In29 : BOOL ;	//Actual value of digi. NCK input 29
   E_ActVal_In30 : BOOL ;	//Actual value of digi. NCK input 30
   E_ActVal_In31 : BOOL ;	//Actual value of digi. NCK input 31
   E_ActVal_In32 : BOOL ;	//Actual value of digi. NCK input 32
   E_ActVal_In33 : BOOL ;	//Actual value of digi. NCK input 33
   E_ActVal_In34 : BOOL ;	//Actual value of digi. NCK input 34
   E_ActVal_In35 : BOOL ;	//Actual value of digi. NCK input 35
   E_ActVal_In36 : BOOL ;	//Actual value of digi. NCK input 36
   E_ActVal_In37 : BOOL ;	//Actual value of digi. NCK input 37
   E_ActVal_In38 : BOOL ;	//Actual value of digi. NCK input 38
   E_ActVal_In39 : BOOL ;	//Actual value of digi. NCK input 39
   E_ActVal_In40 : BOOL ;	//Actual value of digi. NCK input 40
   E_Setpoint_Out9 : BOOL ;	//Setpoint of digi. NCK output 9
   E_Setpoint_Out10 : BOOL ;	//Setpoint of digi. NCK output 10
   E_Setpoint_Out11 : BOOL ;	//Setpoint of digi. NCK output 11
   E_Setpoint_Out12 : BOOL ;	//Setpoint of digi. NCK output 12
   E_Setpoint_Out13 : BOOL ;	//Setpoint of digi. NCK output 13
   E_Setpoint_Out14 : BOOL ;	//Setpoint of digi. NCK output 14
   E_Setpoint_Out15 : BOOL ;	//Setpoint of digi. NCK output 15
   E_Setpoint_Out16 : BOOL ;	//Setpoint of digi. NCK output 16
   E_Setpoint_Out17 : BOOL ;	//Setpoint of digi. NCK output 17
   E_Setpoint_Out18 : BOOL ;	//Setpoint of digi. NCK output 18
   E_Setpoint_Out19 : BOOL ;	//Setpoint of digi. NCK output 19
   E_Setpoint_Out20 : BOOL ;	//Setpoint of digi. NCK output 20
   E_Setpoint_Out21 : BOOL ;	//Setpoint of digi. NCK output 21
   E_Setpoint_Out22 : BOOL ;	//Setpoint of digi. NCK output 22
   E_Setpoint_Out23 : BOOL ;	//Setpoint of digi. NCK output 23
   E_Setpoint_Out24 : BOOL ;	//Setpoint of digi. NCK output 24
   E_Setpoint_Out25 : BOOL ;	//Setpoint of digi. NCK output 25
   E_Setpoint_Out26 : BOOL ;	//Setpoint of digi. NCK output 26
   E_Setpoint_Out27 : BOOL ;	//Setpoint of digi. NCK output 27
   E_Setpoint_Out28 : BOOL ;	//Setpoint of digi. NCK output 28
   E_Setpoint_Out29 : BOOL ;	//Setpoint of digi. NCK output 29
   E_Setpoint_Out30 : BOOL ;	//Setpoint of digi. NCK output 30
   E_Setpoint_Out31 : BOOL ;	//Setpoint of digi. NCK output 31
   E_Setpoint_Out32 : BOOL ;	//Setpoint of digi. NCK output 32
   E_Setpoint_Out33 : BOOL ;	//Setpoint of digi. NCK output 33
   E_Setpoint_Out34 : BOOL ;	//Setpoint of digi. NCK output 34
   E_Setpoint_Out35 : BOOL ;	//Setpoint of digi. NCK output 35
   E_Setpoint_Out36 : BOOL ;	//Setpoint of digi. NCK output 36
   E_Setpoint_Out37 : BOOL ;	//Setpoint of digi. NCK output 37
   E_Setpoint_Out38 : BOOL ;	//Setpoint of digi. NCK output 38
   E_Setpoint_Out39 : BOOL ;	//Setpoint of digi. NCK output 39
   E_Setpoint_Out40 : BOOL ;	//Setpoint of digi. NCK output 40
   E_ActVal_anaIn1 : WORD ;	//Actual value of analog NCK input 1
   E_ActVal_anaIn2 : WORD ;	//Actual value of analog NCK input 2
   E_ActVal_anaIn3 : WORD ;	//Actual value of analog NCK input 3
   E_ActVal_anaIn4 : WORD ;	//Actual value of analog NCK input 4
   E_ActVal_anaIn5 : WORD ;	//Actual value of analog NCK input 5
   E_ActVal_anaIn6 : WORD ;	//Actual value of analog NCK input 6
   E_ActVal_anaIn7 : WORD ;	//Actual value of analog NCK input 7
   E_ActVal_anaIn8 : WORD ;	//Actual value of analog NCK input 8
   E_SetVal_anaOut1 : WORD ;	//Set value of analog NCK output 1
   E_SetVal_anaOut2 : WORD ;	//Set value of analog NCK output 2
   E_SetVal_anaOut3 : WORD ;	//Set value of analog NCK output 3
   E_SetVal_anaOut4 : WORD ;	//Set value of analog NCK output 4
   E_SetVal_anaOut5 : WORD ;	//Set value of analog NCK output 5
   E_SetVal_anaOut6 : WORD ;	//Set value of analog NCK output 6
   E_SetVal_anaOut7 : WORD ;	//Set value of analog NCK output 7
   E_SetVal_anaOut8 : WORD ;	//Set value of analog NCK output 8
   E_CollCheck : ARRAY  [0 .. 7 ] OF BYTE ;	//CollisionsCheck
   A_CollCheck : ARRAY  [0 .. 7 ] OF BYTE ;	//CollisionsCheck
  END_STRUCT ;	
BEGIN
   MCP1AxisTbl[1] := B#16#1;
   MCP1AxisTbl[2] := B#16#2;
   MCP1AxisTbl[3] := B#16#3;
   MCP1AxisTbl[4] := B#16#4;
   MCP1AxisTbl[5] := B#16#5;
   MCP1AxisTbl[6] := B#16#6;
   MCP1AxisTbl[7] := B#16#7;
   MCP1AxisTbl[8] := B#16#8;
   MCP1AxisTbl[9] := B#16#9;
   MCP1AxisTbl[10] := B#16#A;
   MCP1AxisTbl[11] := B#16#B;
   MCP1AxisTbl[12] := B#16#C;
   MCP2AxisTbl[1] := B#16#1;
   MCP2AxisTbl[2] := B#16#2;
   MCP2AxisTbl[3] := B#16#3;
   MCP2AxisTbl[4] := B#16#4;
   MCP2AxisTbl[5] := B#16#5;
   MCP2AxisTbl[6] := B#16#6;
   MCP2AxisTbl[7] := B#16#7;
   MCP2AxisTbl[8] := B#16#8;
   MCP2AxisTbl[9] := B#16#9;
   MCP2AxisTbl[10] := B#16#A;
   MCP2AxisTbl[11] := B#16#B;
   MCP2AxisTbl[12] := B#16#C;
END_DATA_BLOCK

DATA_BLOCK "BAG"	// DB 11
VERSION : 0.1
  STRUCT
   A_AUTO : BOOL ;	//AUTOMATIC mode
   A_MDA : BOOL ;	//MDA mode
   A_JOG : BOOL ;	//JOG mode
   f0_3 : BOOL ;
   A_MCDisable : BOOL ;	//Mode change disable
   A_MGStop : BOOL ;	//Mode group stop
   A_MGStopASp : BOOL ;	//Mode group stop axes plus spindle
   A_MGReset : BOOL ;	//Mode group reset
   A_TEACHIN : BOOL ;	//Machine function TEACH IN
   A_REPOS : BOOL ;	//Machine function REPOS
   A_REF : BOOL ;	//Machine function REF
   f1_3 : BOOL ;
   f1_4 : BOOL ;
   f1_5 : BOOL ;
   A_SingleBlock_B : BOOL ;	// Single block type B
   A_SingleBlock_A : BOOL ;	// Single block type A
   A_INC1 : BOOL ;	//INC1
   A_INC10 : BOOL ;	//INC10
   A_INC100 : BOOL ;	//INC100
   A_INC1000 : BOOL ;	//INC1000
   A_INC10000 : BOOL ;	//INC10000
   A_INCVar : BOOL ;	//INC variable
   f3 : BYTE ;
   E_MMC_AUTO : BOOL ;	//MMC Strobe AUTOMATIC mode
   E_MMC_MDA : BOOL ;	//MMC Strobe MDA mode
   E_MMC_JOG : BOOL ;	//MMC Strobe JOG mode
   f4_3 : BOOL ;
   f4_4 : BOOL ;
   f4_5 : BOOL ;
   f4_6 : BOOL ;
   f4_7 : BOOL ;
   E_MMC_TEACHIN : BOOL ;	//MMC Strobe machine function TEACH IN
   E_MMC_REPOS : BOOL ;	//MMC Strobe machine function REPOS
   E_MMC_REF : BOOL ;	//MMC Strobe Machine function REF
   f5_3 : BOOL ;
   f5_4 : BOOL ;
   f5_5 : BOOL ;
   f5_6 : BOOL ;
   f5_7 : BOOL ;
   E_AUTO : BOOL ;	//Active AUTOMATIC mode
   E_MDA : BOOL ;	//Active MDA mode
   E_JOG : BOOL ;	//Active JOG mode
   E_MGOK : BOOL ;	//Mode group ready
   E_MGreseted : BOOL ;	// Mode Group reseted
   E_NCKintJOG : BOOL ;	// NCK internal JOG active
   f6_6 : BOOL ;
   E_ChanReset : BOOL ;	//All channels in reset state
   E_TEACHIN : BOOL ;	//Active machine function TEACH IN
   E_REPOS : BOOL ;	//Active machine function REPOS
   E_REF : BOOL ;	//Active Machine function REF
   f7_3 : BOOL ;
   f7_4 : BOOL ;
   f7_5 : BOOL ;
   f7_6 : BOOL ;
   f7_7 : BOOL ;
   E_INC1 : BOOL ;	//INC1
   E_INC10 : BOOL ;	//INC10
   E_INC100 : BOOL ;	//INC100
   E_INC1000 : BOOL ;	//INC1000
   E_INC10000 : BOOL ;	//INC10000
   E_INCVar : BOOL ;	//INC variable
   f8_6 : BOOL ;
   f8_7 : BOOL ;
   f9 : BYTE ;
   f10 : ARRAY  [10 .. 19 ] OF BYTE ;
   MG : ARRAY  [2 .. 10 ] OF STRUCT
    A_AUTO : BOOL ;	//AUTOMATIC mode
    A_MDA : BOOL ;	//MDA mode
    A_JOG : BOOL ;	//JOG mode
    f0_3 : BOOL ;
    A_MCDisable : BOOL ;	//Mode change disable
    A_MGStop : BOOL ;	//Mode group stop
    A_MGStopASp : BOOL ;	//Mode group stop axes plus spindle
    A_MGReset : BOOL ;	//Mode group reset
    A_TEACHIN : BOOL ;	//Machine function TEACH IN
    A_REPOS : BOOL ;	//Machine function REPOS
    A_REF : BOOL ;	//Machine function REF
    f1_3 : BOOL ;
    f1_4 : BOOL ;
    f1_5 : BOOL ;
    A_SingleBlock_B : BOOL ;	// Single block type B
    A_SingleBlock_A : BOOL ;	// Single block type A
    A_INC1 : BOOL ;	//INC1
    A_INC10 : BOOL ;	//INC10
    A_INC100 : BOOL ;	//INC100
    A_INC1000 : BOOL ;	//INC1000
    A_INC10000 : BOOL ;	//INC10000
    A_INCVar : BOOL ;	//INC variable
    f3 : BYTE ;
    E_MMC_AUTO : BOOL ;	//MMC Strobe AUTOMATIC mode
    E_MMC_MDA : BOOL ;	//MMC Strobe MDA mode
    E_MMC_JOG : BOOL ;	//MMC Strobe JOG mode
    f4_3 : BOOL ;
    f4_4 : BOOL ;
    f4_5 : BOOL ;
    f4_6 : BOOL ;
    f4_7 : BOOL ;
    E_MMC_TEACHIN : BOOL ;	//MMC Strobe machine function TEACH IN
    E_MMC_REPOS : BOOL ;	//MMC Strobe machine function REPOS
    E_MMC_REF : BOOL ;	//MMC Strobe Machine function REF
    f5_3 : BOOL ;
    f5_4 : BOOL ;
    f5_5 : BOOL ;
    f5_6 : BOOL ;
    f5_7 : BOOL ;
    E_AUTO : BOOL ;	//Active AUTOMATIC mode
    E_MDA : BOOL ;	//Active MDA mode
    E_JOG : BOOL ;	//Active JOG mode
    E_MGOK : BOOL ;	//Mode group ready
    E_MGreseted : BOOL ;	// Mode Group reseted
    E_NCKintJOG : BOOL ;	// NCK internal JOG active
    f6_6 : BOOL ;
    E_ChanReset : BOOL ;	//All channels in reset state
    E_TEACHIN : BOOL ;	//Active machine function TEACH IN
    E_REPOS : BOOL ;	//Active machine function REPOS
    E_REF : BOOL ;	//Active machine function REF
    f7_3 : BOOL ;
    f7_4 : BOOL ;
    f7_5 : BOOL ;
    f7_6 : BOOL ;
    f7_7 : BOOL ;
    E_INC1 : BOOL ;	//INC1
    E_INC10 : BOOL ;	//INC10
    E_INC100 : BOOL ;	//INC100
    E_INC1000 : BOOL ;	//INC1000
    E_INC10000 : BOOL ;	//INC10000
    E_INCVar : BOOL ;	//INC variable
    f8_6 : BOOL ;
    f8_7 : BOOL ;
    f9 : BYTE ;
    f10 : ARRAY  [10 .. 19 ] OF BYTE ;
   END_STRUCT ;
  END_STRUCT ;	
BEGIN
END_DATA_BLOCK

DATA_BLOCK DB 15
AUTHOR : NUMERIK
FAMILY : _800D
NAME : Bas_Com
VERSION : 1.5
  STRUCT
   fifoFull : BOOL ;
   readOffset : BYTE ;
   writeOffset : BYTE ;
   filler : BYTE ;
   Fifo : ARRAY  [1 .. 10 ] OF BYTE ;
   pduRefArr : ARRAY  [1 .. 12 ] OF //Little Endian Werte
   STRUCT
    diNo : WORD ;
    diPartLen : WORD ;
    PdiBeg : DWORD ;
   END_STRUCT ;
  END_STRUCT ;	
BEGIN
END_DATA_BLOCK

// DB 16: know-how protected block, not included

DATA_BLOCK "SPL"	// DB 18
TITLE = SPL dataarea
AUTHOR : NUMERIK
FAMILY : _800D
NAME : Basics
VERSION : 1.5
  STRUCT
   INSEP_VALID : ARRAY  [1 .. 8 ] OF BOOL ;	//used external SPL-Inputbytes(HW)
   OUTSEP_VALID : ARRAY  [1 .. 8 ] OF BOOL ;	//used external SPL-Outputbytes(HW)
   INSEP_ADDR : ARRAY  [1 .. 8 ] OF INT ;	//Addresses external SPL-Inputbytes(HW)
   OUTSEP_ADDR : ARRAY  [1 .. 8 ] OF INT ;	//Addresses external SPL-Outputbytes(HW)
   SPL_READY : BOOL ;	//setup finished
   STOP_MODE : BOOL ;	//0= Stop D, 1=Stop E
   SPL_DATA : STRUCT
    INSEP : ARRAY  [1 .. 64 ] OF BOOL ;
    OUTSEP : ARRAY  [1 .. 64 ] OF BOOL ;
    INSIP : ARRAY  [1 .. 64 ] OF BOOL ;
    OUTSIP : ARRAY  [1 .. 64 ] OF BOOL ;
    MARKERSIP : ARRAY  [1 .. 64 ] OF BOOL ;
   END_STRUCT ;
   SPL_DELTA : STRUCT 	//edge difference NCK - PLC for Diagnostic
    INSEP : ARRAY  [1 .. 64 ] OF BOOL ;
    OUTSEP : ARRAY  [1 .. 64 ] OF BOOL ;
    INSIP : ARRAY  [1 .. 64 ] OF BOOL ;
    OUTSIP : ARRAY  [1 .. 64 ] OF BOOL ;
    MARKERSIP : ARRAY  [1 .. 64 ] OF BOOL ;
   END_STRUCT ;
   CMDSI : BOOL ;	//multiplication of Timeout Value by Factor 10
   CMDSI_R1 : BOOL ;	//for future use
   CMDSI_R2 : BOOL ;	//for future use
   CMDSI_R3 : BOOL ;	//for future use
   CMDSI_R4 : BOOL ;	//for future use
   CMDSI_R5 : BOOL ;	//for future use
   CMDSI_R6 : BOOL ;	//for future use
   CMDSI_R7 : BOOL ;	//for future use
   STATUS_R0 : BOOL ;	//for future use
   STATUS_R1 : BOOL ;	//for future use
   STATUS_R2 : BOOL ;	//for future use
   STATUS_R3 : BOOL ;	//for future use
   STATUS_R4 : BOOL ;	//for future use
   COMM_TO : BOOL ;	//Communication Timeout
   STATUS_R6 : BOOL ;	//for future use
   STATUS_R7 : BOOL ;	//for future use
   STATSI : DINT ;	//Status: 0 - no error, 1 - 320 error number
   LEVELSI : DINT ;	//stacklevel SPL-KDV for Diagnostic
   PLCSIOUT : ARRAY  [1 .. 32 ] OF BOOL ;	//Single Channel Signals from NCK
   PLCSIIN : ARRAY  [1 .. 32 ] OF BOOL ;	//Single Channel Signals to NCK
   SPL_STATUS : ARRAY  [1 .. 16 ] OF BOOL ;	//SPL Status from NCK
   INSEP_PROFISAFE : ARRAY  [1 .. 8 ] OF BOOL ;	//external SPL-Inputbytes(HW) with PROFIsafe Slaves
   OUTSEP_PROFISAFE : ARRAY  [1 .. 8 ] OF BOOL ;	//external SPL-Outputbytes(HW) with PROFIsafe Slaves
   NoOfAxisPerBlock : ARRAY  [1 .. 8 ] OF BYTE ;	//Pointer and Tables for Teststop
   BlockPointer : ARRAY  [1 .. 8 ] OF BYTE ;
   AxisTable : ARRAY  [1 .. 31 ] OF BYTE ;
   FSDP : ARRAY  [1 .. 3 ] OF STRUCT
    ERR_REAC : INT ;	// IN: Error reaction
    ERROR : BOOL ;	// OUT: 1=Communication error
    SUBS_ON : BOOL ;	// OUT: 1=Receiver outputs fail-safe values
    DIAG : WORD ;	// OUT: Service information
    RETVAL14 : WORD ;	// OUT: Error code of SFC 14
    RETVAL15 : WORD ;	// OUT: Error code of SFC 15
   END_STRUCT ;
   FRDP : ARRAY  [1 .. 3 ] OF STRUCT
    SUBS : ARRAY  [0 .. 15 ] OF BOOL ;	// IN: Fail-safe value for receive data BOOL 00 ... BOOL 15
    ERR_REAC : INT ;	// IN: Error reaction
    ACK_REI : BOOL ;	// IN: 1=Acknowledgment for reintegration of send data following communication er
    RES1 : BOOL ;	//Reserved
    RES2 : BOOL ;	//Reserved
    RES3 : BOOL ;	//Reserved
    RES4 : BOOL ;	//Reserved
    RES5 : BOOL ;	//Reserved
    RES6 : BOOL ;	//Reserved
    RES7 : BOOL ;	//Reserved
    ERROR : BOOL ;	// OUT: 1=Communication error
    SUBS_ON : BOOL ;	// OUT: 1=Fail-safe values are output
    ACK_REQ : BOOL ;	// OUT: 1=Acknowledgment for reintegration of send data required
    SENDMODE : BOOL ;	// OUT: 1=F_CPU with F_SENDDP in deactivated safety mode
    DIAG : WORD ;	// OUT: Service information
    RETVAL14 : WORD ;	// OUT: Error code of SFC 14
    RETVAL15 : WORD ;	// OUT: Error code of SFC 15
   END_STRUCT ;
  END_STRUCT ;	
BEGIN
END_DATA_BLOCK

DATA_BLOCK "MMC"	// DB 19
VERSION : 0.1
  STRUCT
   A_SCLight : BOOL ;	//Screen light
   A_SCDark : BOOL ;	//Screen darkening
   A_KeyDisable : BOOL ;	//Key disable
   A_ClearCanAl : BOOL ;	//Clear cancel alarms
   A_ClearRecAl : BOOL ;	//Clear recall alarms
   f0_5 : BOOL ;
   f0_6 : BOOL ;
   A_ActWCS : BOOL ;	//Actual value in WCS 0=MCS
   A_1stError1 : WORD ;	//1st error HIGRAPH
   A_1stError2 : WORD ;	//1st error HIGRAPH
   A_ASpi1percent : BYTE ;	//Analog spindle 1:
   A_ASpi2percent : BYTE ;
   A_MCPChan : BYTE ;
   A_OEM1 : BOOL ;
   A_OEM2 : BOOL ;
   A_AToolMeas : BOOL ;	//AutoToolMeasure
   f9_3 : BOOL ;
   f9_4 : BOOL ;
   f9_5 : BOOL ;
   f9_6 : BOOL ;
   f9_7 : BOOL ;
   A_Hardkey : BYTE ;	//PLC Hardkeys
   f11 : BYTE ;	//Reserved for hardkeys
   f12_0 : BOOL ;
   f12_1 : BOOL ;
   A_COM2 : BOOL ;
   A_COM1 : BOOL ;
   A_V24stop : BOOL ;
   A_V24ext : BOOL ;
   A_V24off : BOOL ;
   A_V24on : BOOL ;
   A_TeachDisable : BOOL ;
   f13_1 : BOOL ;
   f13_2 : BOOL ;
   f13_3 : BOOL ;
   f13_4 : BOOL ;
   A_PPdeload : BOOL ;
   A_PPload : BOOL ;
   A_PPsel : BOOL ;
   A_V24Index1 : BYTE ;
   A_V24Index2 : BYTE ;
   A_V24NoFile1 : BYTE ;
   A_V24NoFile2 : BYTE ;
   A_res18 : BYTE ;
   A_res19 : BYTE ;	//Message counter
   f20_0 : BOOL ;
   E_SCDark : BOOL ;	//Screen darkening
   E_Cancel : BOOL ;	//Cancel
   E_CanCleared : BOOL ;	//Cancel alarms cleared
   E_RecCleared : BOOL ;	//Recall alarms cleared
   f20_5 : BOOL ;	//res. Language
   E_SimActiv : BOOL ;	//Simulation active
   E_ActWCS : BOOL ;	//Switchover MCS/WCS 0=MCS
   E_ActivWA : BYTE ;
   E_Chan : BYTE ;	//Channel displayed
   f23 : BYTE ;
   E_V24Err : BOOL ;
   E_V24OK : BOOL ;
   E_V24COM2 : BOOL ;
   E_V24COM1 : BOOL ;
   E_V24stop : BOOL ;
   E_V24ext : BOOL ;
   E_V24off : BOOL ;
   E_V24on : BOOL ;
   E_V24Error : BYTE ;	//V24: Error Byte
   E_res26_0 : BOOL ;	//Reserved
   E_PPOK : BOOL ;	//Part program status OK
   E_PPErr : BOOL ;	//Part program status Error
   E_PPAct : BOOL ;	//Part program status active
   f26_4 : BOOL ;	//Reserved
   E_PPdeload : BOOL ;	//Part program status deloading
   E_PPload : BOOL ;	//Part program status loading
   E_PPsel : BOOL ;	//Part program status selecting
   E_PPError : BYTE ;	//Part program status Error
   A_PictNo : INT ;
   A_PictOn : BOOL ;
   A_PictOff : BOOL ;
   f30_2 : BOOL ;
   f30_3 : BOOL ;
   f30_4 : BOOL ;
   f30_5 : BOOL ;
   f30_6 : BOOL ;
   f30_7 : BOOL ;
   E_PictOK : BOOL ;
   E_PictOn : BOOL ;
   E_PictAct : BOOL ;
   E_PictOff : BOOL ;
   E_PictErr : BOOL ;
   f31_5 : BOOL ;
   f31_6 : BOOL ;
   E_NotAct : BOOL ;
   A_FuncNo : BYTE ;
   A_Par1 : BYTE ;
   A_Par2 : BYTE ;
   A_Par3 : BYTE ;
   E_FuncErr : BYTE ;
   f37 : BYTE ;
   f38 : BYTE ;
   f39 : BYTE ;
   res40 : ARRAY  [0 .. 9 ] OF BYTE ;
   MMC2 : STRUCT
    A_SCLight : BOOL ;	//Screen light
    A_SCDark : BOOL ;	//Screen darkening
    A_KeyDisable : BOOL ;	//Key disable
    A_ClearCanAl : BOOL ;	//Clear cancel alarms
    A_ClearRecAl : BOOL ;	//Clear recall alarms
    f0_5 : BOOL ;
    f0_6 : BOOL ;
    A_ActWCS : BOOL ;	//Actual value in WCS 0=MCS
    A_1stError1 : WORD ;	//1st error HIGRAPH
    A_1stError2 : WORD ;	//1st error HIGRAPH
    A_ASpi1percent : BYTE ;	//Analog spindle 1:
    A_ASpi2percent : BYTE ;
    A_MCPChan : BYTE ;
    A_OEM1 : BOOL ;
    A_OEM2 : BOOL ;
    A_AToolMeas : BOOL ;	//AutoToolMeasure
    f9_3 : BOOL ;
    f9_4 : BOOL ;
    f9_5 : BOOL ;
    f9_6 : BOOL ;
    f9_7 : BOOL ;
    A_Hardkey : BYTE ;	//PLC Hardkeys
    f11 : BYTE ;	//Reserved for hardkeys
    f12_0 : BOOL ;
    f12_1 : BOOL ;
    A_COM2 : BOOL ;
    A_COM1 : BOOL ;
    A_V24stop : BOOL ;
    A_V24ext : BOOL ;
    A_V24off : BOOL ;
    A_V24on : BOOL ;
    f13_0 : BOOL ;
    f13_1 : BOOL ;
    f13_2 : BOOL ;
    f13_3 : BOOL ;
    f13_4 : BOOL ;
    A_PPdeload : BOOL ;
    A_PPload : BOOL ;
    A_PPsel : BOOL ;
    A_V24Index1 : BYTE ;
    A_V24Index2 : BYTE ;
    A_V24NoFile1 : BYTE ;
    A_V24NoFile2 : BYTE ;
    A_res18 : BYTE ;
    A_res19 : BYTE ;	//Message counter
    f20_0 : BOOL ;
    E_SCDark : BOOL ;	//Screen darkening
    E_Cancel : BOOL ;	//Cancel
    E_CanCleared : BOOL ;	//Cancel alarms cleared
    E_RecCleared : BOOL ;	//Recall alarms cleared
    f20_5 : BOOL ;	//res. Language
    E_SimActiv : BOOL ;	//Simulation active
    E_ActWCS : BOOL ;	//Switchover MCS/WCS 0=MCS
    E_ActivWA : BYTE ;
    E_Chan : BYTE ;	//Channel displayed
    f23 : BYTE ;
    E_V24Err : BOOL ;
    E_V24OK : BOOL ;
    E_V24COM2 : BOOL ;
    E_V24COM1 : BOOL ;
    E_V24stop : BOOL ;
    E_V24ext : BOOL ;
    E_V24off : BOOL ;
    E_V24on : BOOL ;
    E_V24Error : BYTE ;	//V24: Error Byte
    E_res26_0 : BOOL ;	//Reserved
    E_PPOK : BOOL ;	//Part program status OK
    E_PPErr : BOOL ;	//Part program status Error
    E_PPAct : BOOL ;	//Part program status active
    f26_4 : BOOL ;	//Reserved
    E_PPdeload : BOOL ;	//Part program status deloading
    E_PPload : BOOL ;	//Part program status loading
    E_PPsel : BOOL ;	//Part program status selecting
    E_PPError : BYTE ;	//Part program status Error
    A_PictNo : INT ;
    A_PictOn : BOOL ;
    A_PictOff : BOOL ;
    f30_2 : BOOL ;
    f30_3 : BOOL ;
    f30_4 : BOOL ;
    f30_5 : BOOL ;
    f30_6 : BOOL ;
    f30_7 : BOOL ;
    E_PictOK : BOOL ;
    E_PictOn : BOOL ;
    E_PictAct : BOOL ;
    E_PictOff : BOOL ;
    E_PictErr : BOOL ;
    f31_5 : BOOL ;
    f31_6 : BOOL ;
    E_NotAct : BOOL ;
    A_FuncNo : BYTE ;
    A_Par1 : BYTE ;
    A_Par2 : BYTE ;
    A_Par3 : BYTE ;
    E_FuncErr : BYTE ;
    f37 : BYTE ;
    f38 : BYTE ;
    f39 : BYTE ;
    res40 : ARRAY  [0 .. 9 ] OF BYTE ;
   END_STRUCT ;	//M to N
   ONL_REQUEST : WORD ;
   ONL_CONFIRM : WORD ;
   PAR_CLIENT_IDENT : WORD ;
   PAR_MMC_TYP : BYTE ;
   PAR_MSTT_ADR : BYTE ;
   PAR_STATUS : BYTE ;
   PAR_Z_INFO : BYTE ;
   MtoNAlive : WORD ;
   f112 : BYTE ;
   ParOpKeyAdr : BYTE ;
   ParTcuIndex : BYTE ;
   f115 : BYTE ;
   Tcu1KeyAdr : BYTE ;
   Tcu2KeyAdr : BYTE ;
   Tcu1Index : BYTE ;
   Tcu2Index : BYTE ;
   MMC1_CLIENT_IDENT : WORD ;
   MMC1_TYP : BYTE ;
   MMC1_MSTT_ADR : BYTE ;
   MMC1_STATUS : BYTE ;
   MMC1_Z_INFO : BYTE ;
   MMC1_SHIFT_LOCK : BOOL ;
   MMC1_MSTT_SHIFT_LOCK : BOOL ;
   MMC1_ACTIVE_REQ : BOOL ;
   MMC1_ACTIVE_PERM : BOOL ;
   MMC1_ACTIVE_CHANGED : BOOL ;
   MMC1_CHANGED_DENIED : BOOL ;
   MMC1_TCU_SHIFT_LOCK : BOOL ;
   f127 : BYTE ;
   MMC1_TRANS_DB : WORD ;
   MMC2_CLIENT_IDENT : WORD ;
   MMC2_TYP : BYTE ;
   MMC2_MSTT_ADR : BYTE ;
   MMC2_STATUS : BYTE ;
   MMC2_Z_INFO : BYTE ;
   MMC2_SHIFT_LOCK : BOOL ;
   MMC2_MSTT_SHIFT_LOCK : BOOL ;
   MMC2_ACTIVE_REQ : BOOL ;
   MMC2_ACTIVE_PERM : BOOL ;
   MMC2_ACTIVE_CHANGED : BOOL ;
   MMC2_CHANGED_DENIED : BOOL ;
   MMC2_TCU_SHIFT_LOCK : BOOL ;
   f137 : BYTE ;
   MMC2_TRANS_DB : WORD ;
   A_Subtype : INT ;	//for Codecarrier Input from PLC
   A_Duplo : INT ;
   A_Ident : STRING  [32 ];
   A_Tnumber : INT ;
   A_MagazinePlace : INT ;
   A_MagazinePlaceType : INT ;
   A_ToolSize_Upper : BYTE ;
   A_ToolSize_Down : BYTE ;
   A_ToolSize_Left : BYTE ;
   A_ToolSize_Right : BYTE ;
   A_Channel : BYTE ;
   A_LoadingPlace : BYTE ;
   A_Magazine : INT ;
   A_Unit : BYTE ;
   A_NCU_Index : BYTE ;
   A_FileIndex : INT ;
   A_ActiveEnable : BOOL ;
   A_Override : BOOL ;
   A_LoadTool : BOOL ;
   A_DeleteTool : BOOL ;
   E_Subtype : INT ;	//for Codecarrier Output to PLC
   E_Duplo : INT ;
   E_Ident : STRING  [32 ];
   E_Tnumber : INT ;
   E_ToolState : INT ;
   E_MagazinePlaceType : INT ;
   E_ToolSize_Upper : BYTE ;
   E_ToolSize_Down : BYTE ;
   E_ToolSize_Left : BYTE ;
   E_ToolSize_Right : BYTE ;
   E_Magazine : INT ;
   E_MagazinePlace : INT ;
   A_ReqMMC1 : BOOL ;	//for Codecarrier Request MMC-Interface1
   A_ReqMMC2 : BOOL ;	//for Codecarrier Request MMC-Interface2
   A_K_Code : BYTE ;
   E_Done : BOOL ;
   E_Error : BOOL ;
   E_Active : BOOL ;	// CodeCarrierReadEnable : BOOL;
// CodeCarrierWriteEnable : BOOL;
   E_K_CodeError : BYTE ;	//Identify for Error_Code
   E_Error_Code : INT ;
   E_Req : BOOL ;	//for Positioning
   f257 : BYTE ;
   A_Done : BOOL ;
   A_Error : BOOL ;
   A_Active : BOOL ;
   f258_3 : BOOL ;
   f258_4 : BOOL ;
   f258_5 : BOOL ;
   f258_6 : BOOL ;
   f258_7 : BOOL ;
   E_TDC_Read : BOOL ;
   E_TDC_Write : BOOL ;
   E_TDC_Cancel : BOOL ;
   A_Error_Code : INT ;
   E_PMagazine : INT ;
   E_PMagazinePlace : INT ;
   E_PTnumber : INT ;	//TPM-Data
   A_TPMStatus : INT ;
   A_TPMCounter : ARRAY  [1 .. 32 ] OF DINT ;
  END_STRUCT ;	
BEGIN
END_DATA_BLOCK

